(* LS Electric XG5000 project: 210109_AX_FRT_FLR *)
(* PLC NewPLC *)
(* module base 0 slot 0: FEnet:XGL-EFMT(B) (Fast Ethernet 통신 모듈, 전기 Master) *)
(* module base 0 slot 1: FEnet:XGL-EFMT(B) (Fast Ethernet 통신 모듈, 전기 Master) *)
(* module base 0 slot 2: FEnet:XGL-EFMT(B) (Fast Ethernet 통신 모듈, 전기 Master) *)
(* module base 0 slot 3: FEnet:XGL-EFMT(B) (Fast Ethernet 통신 모듈, 전기 Master) *)
(* module base 0 slot 4: FEnet:XGL-EFMT(B) (Fast Ethernet 통신 모듈, 전기 Master) *)
(* module base 0 slot 5: FEnet:XGL-EFMT(B) (Fast Ethernet 통신 모듈, 전기 Master) *)
(* module base 0 slot 6: FEnet:XGL-EFMT(B) (Fast Ethernet 통신 모듈, 전기 Master) *)
(* module base 0 slot 7: FEnet:XGL-EFMT(B) (Fast Ethernet 통신 모듈, 전기 Master) *)
(* module base 0 slot 0: 입력 모듈:XBE-DC16A/B (DC24V 입력, 16점 / DC12/24V 입력, 16점) *)
(* module base 0 slot 1: 입력 모듈:XBE-DC16A/B (DC24V 입력, 16점 / DC12/24V 입력, 16점) *)
(* module base 0 slot 2: 입력 모듈:XBE-DC16A/B (DC24V 입력, 16점 / DC12/24V 입력, 16점) *)
(* module base 0 slot 3: 입력 모듈:XBE-DC16A/B (DC24V 입력, 16점 / DC12/24V 입력, 16점) *)
(* module base 0 slot 4: 출력 모듈:XBE-TN/TP16A (트랜지스터 출력, 16점 (싱크출력/소스출력)) *)
(* module base 0 slot 5: 출력 모듈:XBE-TN/TP16A (트랜지스터 출력, 16점 (싱크출력/소스출력)) *)
(* module base 0 slot 6: 출력 모듈:XBE-TN/TP16A (트랜지스터 출력, 16점 (싱크출력/소스출력)) *)
(* module base 0 slot 7: 출력 모듈:XBE-TN/TP16A (트랜지스터 출력, 16점 (싱크출력/소스출력)) *)
(* module base 0 slot 0: 입력 모듈:XBE-DC16A/B (DC24V 입력, 16점 / DC12/24V 입력, 16점) *)
(* module base 0 slot 1: 입력 모듈:XBE-DC16A/B (DC24V 입력, 16점 / DC12/24V 입력, 16점) *)
(* module base 0 slot 2: 입력 모듈:XBE-DC16A/B (DC24V 입력, 16점 / DC12/24V 입력, 16점) *)
(* module base 0 slot 3: 출력 모듈:XBE-TN/TP16A (트랜지스터 출력, 16점 (싱크출력/소스출력)) *)
(* module base 0 slot 4: 출력 모듈:XBE-TN/TP16A (트랜지스터 출력, 16점 (싱크출력/소스출력)) *)
(* module base 0 slot 0: 입력 모듈:XBE-DC16A/B (DC24V 입력, 16점 / DC12/24V 입력, 16점) *)
(* module base 0 slot 1: 입력 모듈:XBE-DC16A/B (DC24V 입력, 16점 / DC12/24V 입력, 16점) *)
(* module base 0 slot 2: 입력 모듈:XBE-DC16A/B (DC24V 입력, 16점 / DC12/24V 입력, 16점) *)
(* module base 0 slot 3: 출력 모듈:XBE-TN/TP16A (트랜지스터 출력, 16점 (싱크출력/소스출력)) *)
(* module base 0 slot 4: 출력 모듈:XBE-TN/TP16A (트랜지스터 출력, 16점 (싱크출력/소스출력)) *)
(* module base 0 slot 0: 입력 모듈:XBE-DC16A/B (DC24V 입력, 16점 / DC12/24V 입력, 16점) *)
(* module base 0 slot 1: 입력 모듈:XBE-DC16A/B (DC24V 입력, 16점 / DC12/24V 입력, 16점) *)
(* module base 0 slot 2: 입력 모듈:XBE-DC16A/B (DC24V 입력, 16점 / DC12/24V 입력, 16점) *)
(* module base 0 slot 3: 출력 모듈:XBE-TN/TP16A (트랜지스터 출력, 16점 (싱크출력/소스출력)) *)
(* module base 0 slot 4: 출력 모듈:XBE-TN/TP16A (트랜지스터 출력, 16점 (싱크출력/소스출력)) *)
(* module base 0 slot 0: 입력 모듈:XBE-DC16A/B (DC24V 입력, 16점 / DC12/24V 입력, 16점) *)
(* module base 0 slot 1: 출력 모듈:XBE-TN/TP16A (트랜지스터 출력, 16점 (싱크출력/소스출력)) *)
(* module base 0 slot 2: 입력 모듈:XBE-DC16A/B (DC24V 입력, 16점 / DC12/24V 입력, 16점) *)
(* module base 0 slot 3: 출력 모듈:XBE-TN/TP16A (트랜지스터 출력, 16점 (싱크출력/소스출력)) *)
(* module base 0 slot 0: 입력 모듈:XBE-DC16A/B (DC24V 입력, 16점 / DC12/24V 입력, 16점) *)
(* module base 0 slot 1: 입력 모듈:XBE-DC16A/B (DC24V 입력, 16점 / DC12/24V 입력, 16점) *)
(* module base 0 slot 2: 출력 모듈:XBE-TN/TP16A (트랜지스터 출력, 16점 (싱크출력/소스출력)) *)
(* module base 0 slot 3: 입력 모듈:XBE-DC16A/B (DC24V 입력, 16점 / DC12/24V 입력, 16점) *)
(* module base 0 slot 4: 출력 모듈:XBE-TN/TP16A (트랜지스터 출력, 16점 (싱크출력/소스출력)) *)
(* module base 0 slot 0: 입력 모듈:XBE-DC16A/B (DC24V 입력, 16점 / DC12/24V 입력, 16점) *)
(* module base 0 slot 1: 입력 모듈:XBE-DC16A/B (DC24V 입력, 16점 / DC12/24V 입력, 16점) *)
(* module base 0 slot 2: 출력 모듈:XBE-TN/TP16A (트랜지스터 출력, 16점 (싱크출력/소스출력)) *)
(* module base 0 slot 3: 입력 모듈:XBE-DC16A/B (DC24V 입력, 16점 / DC12/24V 입력, 16점) *)
(* module base 0 slot 4: 출력 모듈:XBE-TN/TP16A (트랜지스터 출력, 16점 (싱크출력/소스출력)) *)
(* module base 0 slot 0: 입력 모듈:XBE-DC16A/B (DC24V 입력, 16점 / DC12/24V 입력, 16점) *)
(* module base 0 slot 1: 입력 모듈:XBE-DC16A/B (DC24V 입력, 16점 / DC12/24V 입력, 16점) *)
(* module base 0 slot 2: 입력 모듈:XBE-DC16A/B (DC24V 입력, 16점 / DC12/24V 입력, 16점) *)
(* module base 0 slot 3: 출력 모듈:XBE-TN/TP16A (트랜지스터 출력, 16점 (싱크출력/소스출력)) *)
(* module base 0 slot 4: 출력 모듈:XBE-TN/TP16A (트랜지스터 출력, 16점 (싱크출력/소스출력)) *)
(* module base 0 slot 5: 입력 모듈:XBE-DC16A/B (DC24V 입력, 16점 / DC12/24V 입력, 16점) *)
(* module base 0 slot 6: 출력 모듈:XBE-TN/TP16A (트랜지스터 출력, 16점 (싱크출력/소스출력)) *)
VAR_GLOBAL
    APRON_LH_RACK1_I_막장감지 AT %MW87211.2 : BOOL;
    APRON_LH_RACK1_I_종발이감지1 AT %MW87211.0 : BOOL;
    APRON_LH_RACK1_I_종발이감지2 AT %MW87211.1 : BOOL;
    APRON_LH_RACK2_I_막장감지 AT %MW87211.10 : BOOL;
    APRON_LH_RACK2_I_종발이감지1 AT %MW87211.8 : BOOL;
    APRON_LH_RACK2_I_종발이감지2 AT %MW87211.9 : BOOL;
    APRON_RH_RACK1_I_막장감지 AT %MW87210.2 : BOOL;
    APRON_RH_RACK1_I_종발이감지1 AT %MW87210.0 : BOOL;
    APRON_RH_RACK1_I_종발이감지2 AT %MW87210.1 : BOOL;
    APRON_RH_RACK2_I_막장감지 AT %MW87210.10 : BOOL;
    APRON_RH_RACK2_I_종발이감지1 AT %MW87210.8 : BOOL;
    APRON_RH_RACK2_I_종발이감지2 AT %MW87210.9 : BOOL;
    AWAYS_OFF AT %MW3.0 : BOOL;
    AWAYS_ON AT %MW3.1 : BOOL;
    CARTYPE AT %MW10000 : ARRAY[0..999] OF WORD; (* CARTYPE *)
    CLOCK_BIT_0_1Sec AT %MW0.0 : BOOL;
    CLOCK_BIT_0_2Sec AT %MW0.1 : BOOL;
    CLOCK_BIT_0_4Sec AT %MW0.2 : BOOL;
    CLOCK_BIT_0_5Sec AT %MW0.3 : BOOL;
    CLOCK_BIT_0_8Sec AT %MW0.4 : BOOL;
    CLOCK_BIT_1_0Sec AT %MW0.5 : BOOL;
    CLOCK_BIT_1_6Sec AT %MW0.6 : BOOL;
    CLOCK_BIT_2_0Sec AT %MW0.7 : BOOL;
    DASH_RACK1_I_막장감지 AT %MW87300.2 : BOOL;
    DASH_RACK1_I_종발이감지1 AT %MW87300.0 : BOOL;
    DASH_RACK1_I_종발이감지2 AT %MW87300.1 : BOOL;
    DASH_RACK2_I_막장감지 AT %MW87300.10 : BOOL;
    DASH_RACK2_I_종발이감지1 AT %MW87300.8 : BOOL;
    DASH_RACK2_I_종발이감지2 AT %MW87300.9 : BOOL;
    DASH_RACK3_I_막장감지 AT %MW87301.2 : BOOL;
    DASH_RACK3_I_종발이감지1 AT %MW87301.0 : BOOL;
    DASH_RACK3_I_종발이감지2 AT %MW87301.1 : BOOL;
    DASH_RACK4_I_막장감지 AT %MW87301.10 : BOOL;
    DASH_RACK4_I_종발이감지1 AT %MW87301.8 : BOOL;
    DASH_RACK4_I_종발이감지2 AT %MW87301.9 : BOOL;
    EGIS_EJS : BOOL;
    F_COMPL_I_CYCLE_정지_OK AT %MW83211.7 : BOOL;
    F_COMPL_I_SAFTY_이상 AT %MW83210.14 : BOOL;
    F_COMPL_I_SP1 AT %MW83210.4 : BOOL;
    F_COMPL_I_SP10 AT %MW83211.8 : BOOL;
    F_COMPL_I_SP11 AT %MW83211.9 : BOOL;
    F_COMPL_I_SP12 AT %MW83211.10 : BOOL;
    F_COMPL_I_SP13 AT %MW83211.11 : BOOL;
    F_COMPL_I_SP14 AT %MW83211.12 : BOOL;
    F_COMPL_I_SP15 AT %MW83211.13 : BOOL;
    F_COMPL_I_SP16 AT %MW83211.14 : BOOL;
    F_COMPL_I_SP2 AT %MW83210.5 : BOOL;
    F_COMPL_I_SP3 AT %MW83210.6 : BOOL;
    F_COMPL_I_SP4 AT %MW83210.7 : BOOL;
    F_COMPL_I_SP7 AT %MW83210.10 : BOOL;
    F_COMPL_I_SP8 AT %MW83210.11 : BOOL;
    F_COMPL_I_SP9 AT %MW83210.12 : BOOL;
    F_COMPL_I_SPARE_진입OK AT %MW83211.2 : BOOL;
    F_COMPL_I_도착완료 AT %MW83211.6 : BOOL;
    F_COMPL_I_불간섭 AT %MW83211.0 : BOOL;
    F_COMPL_I_비상정지 AT %MW83210.15 : BOOL;
    F_COMPL_I_수동모드 AT %MW83210.1 : BOOL;
    F_COMPL_I_운전준비 AT %MW83210.0 : BOOL;
    F_COMPL_I_자동_운전중 AT %MW83210.3 : BOOL;
    F_COMPL_I_자동모드 AT %MW83210.2 : BOOL;
    F_COMPL_I_작업완료 AT %MW83211.5 : BOOL;
    F_COMPL_I_진입OK AT %MW83211.1 : BOOL;
    F_COMPL_I_차종수신완료 AT %MW83211.4 : BOOL;
    F_COMPL_I_차종요구 AT %MW83211.3 : BOOL;
    F_COMPL_I_총괄_이상 AT %MW83210.13 : BOOL;
    F_COMPL_I_통신_CHK AT %MW83211.15 : BOOL;
    F_COMPL_I_파트_NONE AT %MW83210.9 : BOOL;
    F_COMPL_I_파트_ON AT %MW83210.8 : BOOL;
    F_COMPL_O_1차종_2차종_3차종 AT %MW93221 : WORD;
    F_COMPL_O_4차종 AT %MW93222 : WORD;
    F_COMPL_O_5차종_6차종_7차종 AT %MW93223 : WORD;
    F_COMPL_O_8차종_9차종 AT %MW93224 : WORD;
    F_COMPL_O_CYCLE_정지_OK AT %MW93211.7 : BOOL;
    F_COMPL_O_SAFTY_이상 AT %MW93210.14 : BOOL;
    F_COMPL_O_SEQ_1 AT %MW93220 : WORD;
    F_COMPL_O_SP1 AT %MW93210.4 : BOOL;
    F_COMPL_O_SP10 AT %MW93211.8 : BOOL;
    F_COMPL_O_SP11 AT %MW93211.9 : BOOL;
    F_COMPL_O_SP12 AT %MW93211.10 : BOOL;
    F_COMPL_O_SP13 AT %MW93211.11 : BOOL;
    F_COMPL_O_SP14 AT %MW93211.12 : BOOL;
    F_COMPL_O_SP15 AT %MW93211.13 : BOOL;
    F_COMPL_O_SP16 AT %MW93211.14 : BOOL;
    F_COMPL_O_SP2 AT %MW93210.5 : BOOL;
    F_COMPL_O_SP3 AT %MW93210.6 : BOOL;
    F_COMPL_O_SP4 AT %MW93210.7 : BOOL;
    F_COMPL_O_SP5 AT %MW93210.8 : BOOL;
    F_COMPL_O_SP6 AT %MW93210.9 : BOOL;
    F_COMPL_O_SP7 AT %MW93210.10 : BOOL;
    F_COMPL_O_SP8 AT %MW93210.11 : BOOL;
    F_COMPL_O_SP9 AT %MW93210.12 : BOOL;
    F_COMPL_O_SPARE_진입OK AT %MW93211.2 : BOOL;
    F_COMPL_O_VIN_NO11 AT %MW93229 : WORD;
    F_COMPL_O_VIN_NO12 AT %MW93230 : WORD;
    F_COMPL_O_VIN_NO13 AT %MW93231 : WORD;
    F_COMPL_O_VIN_NO14 AT %MW93232 : WORD;
    F_COMPL_O_VIN_NO15 AT %MW93233 : WORD;
    F_COMPL_O_도착완료 AT %MW93211.6 : BOOL;
    F_COMPL_O_불간섭 AT %MW93211.0 : BOOL;
    F_COMPL_O_비상정지 AT %MW93210.15 : BOOL;
    F_COMPL_O_수동모드 AT %MW93210.1 : BOOL;
    F_COMPL_O_옵션차종1 AT %MW93225 : WORD;
    F_COMPL_O_옵션차종2 AT %MW93226 : WORD;
    F_COMPL_O_옵션차종3 AT %MW93227 : WORD;
    F_COMPL_O_운영정보 AT %MW93228 : WORD;
    F_COMPL_O_운전준비 AT %MW93210.0 : BOOL;
    F_COMPL_O_자동_운전중 AT %MW93210.3 : BOOL;
    F_COMPL_O_자동모드 AT %MW93210.2 : BOOL;
    F_COMPL_O_작업완료 AT %MW93211.5 : BOOL;
    F_COMPL_O_진입OK AT %MW93211.1 : BOOL;
    F_COMPL_O_차종수신완료 AT %MW93211.4 : BOOL;
    F_COMPL_O_차종요구 AT %MW93211.3 : BOOL;
    F_COMPL_O_총괄_이상 AT %MW93210.13 : BOOL;
    F_COMPL_O_통신_CHK AT %MW93211.15 : BOOL;
    GATE10_M_CP_TRIP AT %MW409.15 : BOOL;
    GATE10_M_GATE_OPEN AT %MW409.13 : BOOL;
    GATE10_M_RESTART AT %MW409.1 : BOOL;
    GATE10_M_도어_잠김 AT %MW409.3 : BOOL;
    GATE10_M_비상정지 AT %MW409.7 : BOOL;
    GATE10_M_이상_리셋 AT %MW409.0 : BOOL;
    GATE10_M_정상 AT %MW409.4 : BOOL;
    GATE10_M_정지_CALL AT %MW409.2 : BOOL;
    GATE10_M_통신_이상 AT %MW409.14 : BOOL;
    GATE11_M_CP_TRIP AT %MW410.15 : BOOL;
    GATE11_M_GATE_OPEN AT %MW410.13 : BOOL;
    GATE11_M_RESTART AT %MW410.1 : BOOL;
    GATE11_M_도어_잠김 AT %MW410.3 : BOOL;
    GATE11_M_비상정지 AT %MW410.7 : BOOL;
    GATE11_M_이상_리셋 AT %MW410.0 : BOOL;
    GATE11_M_정상 AT %MW410.4 : BOOL;
    GATE11_M_정지_CALL AT %MW410.2 : BOOL;
    GATE11_M_통신_이상 AT %MW410.14 : BOOL;
    GATE12_M_CP_TRIP AT %MW411.15 : BOOL;
    GATE12_M_GATE_OPEN AT %MW411.13 : BOOL;
    GATE12_M_RESTART AT %MW411.1 : BOOL;
    GATE12_M_도어_잠김 AT %MW411.3 : BOOL;
    GATE12_M_비상정지 AT %MW411.7 : BOOL;
    GATE12_M_이상_리셋 AT %MW411.0 : BOOL;
    GATE12_M_정상 AT %MW411.4 : BOOL;
    GATE12_M_정지_CALL AT %MW411.2 : BOOL;
    GATE12_M_통신_이상 AT %MW411.14 : BOOL;
    GATE_10_M_GATE_OPEN_보조 AT %MW409.12 : BOOL;
    GATE_11_M_GATE_OPEN_보조 AT %MW410.12 : BOOL;
    GATE_12_M_GATE_OPEN_보조 AT %MW411.12 : BOOL;
    GB10_7_10_PLC_BOX_CP_TRIP AT %MW87100.15 : BOOL; (* 입력 접점 15 *)
    GB10_EPB_비상정지1 AT %MW87102.0 : BOOL; (* 입력 접점 00 *)
    GB10_EPB_비상정지2 AT %MW87102.1 : BOOL; (* 입력 접점 01 *)
    GB10_GATE_LOCK_SW_열림1 AT %MW87102.8 : BOOL; (* 입력 접점 08 *)
    GB10_GATE_LOCK_SW_열림2 AT %MW87102.9 : BOOL; (* 입력 접점 09 *)
    GB10_PBL_CYCLE_정지 AT %MW87100.1 : BOOL; (* 입력 접점 01 *)
    GB10_PBL_CYCLE_정지_LP AT %MW97101.1 : BOOL; (* 출력 접점 01 *)
    GB10_PBL_자동_운전 AT %MW87100.0 : BOOL; (* 입력 접점 00 *)
    GB10_PBL_자동_운전_LP AT %MW97101.0 : BOOL; (* 출력 접점 00 *)
    GB10_PB_이상_리셋 AT %MW87100.2 : BOOL; (* 입력 접점 02 *)
    GB10_SAFETY_DOOR_UNLOOK1 AT %MW97103.0 : BOOL; (* 출력 접점 00 *)
    GB10_SAFETY_DOOR_UNLOOK2 AT %MW97103.1 : BOOL; (* 출력 접점 01 *)
    GB10_TL_GREEN_LAMP AT %MW97101.9 : BOOL; (* 출력 접점 09 *)
    GB10_TL_RED_LAMP AT %MW97101.8 : BOOL; (* 출력 접점 08 *)
    HMI_M_SEL_MOD_S101 AT %MW6.1 : BOOL;
    HMI_M_SEL_MOD_S102 AT %MW6.2 : BOOL;
    HMI_M_SEL_MOD_S103 AT %MW6.3 : BOOL;
    HMI_M_SEL_MOD_STN AT %MW6.0 : BOOL;
    HMI_M_매칭_R102_1_S101 AT %MW70.1 : BOOL;
    HMI_M_매칭_S101_R102_1 AT %MW70.0 : BOOL;
    HMI_M_매칭선택 AT %MW70 : WORD;
    HMI_M_매칭차종_DATA_OK AT %MW9.9 : BOOL;
    HMI_M_매칭차종_복사_ON AT %MW9.6 : BOOL;
    HMI_M_매칭차종_복사_SET AT %MW9.8 : BOOL;
    HMI_M_매칭차종_복사_가능 AT %MW9.7 : BOOL;
    HMI_M_선택_MOD_CARR AT %MW12 : WORD;
    HMI_M_선택_MOD_PROF AT %MW13 : WORD;
    HMI_M_차종매칭 AT %MW50 : ARRAY[0..19] OF WORD;
    HMI_M_차종매칭_SEQ AT %MW50 : WORD;
    HMI_M_차종매칭_VIN_NO_1_2 AT %MW61 : WORD;
    HMI_M_차종매칭_VIN_NO_3_4 AT %MW62 : WORD;
    HMI_M_차종매칭_VIN_NO_5_6 AT %MW63 : WORD;
    HMI_M_차종매칭_VIN_NO_7_8 AT %MW64 : WORD;
    HMI_M_차종매칭_VIN_NO_9_10 AT %MW65 : WORD;
    HMI_M_차종매칭_차종1_AX AT %MW51.0 : BOOL;
    HMI_M_차종매칭_차종1_B AT %MW51.1 : BOOL;
    HMI_M_차종매칭_차종1_C AT %MW51.2 : BOOL;
    HMI_M_차종매칭_차종1_D AT %MW51.3 : BOOL;
    HMI_M_차종매칭_차종1_E AT %MW51.4 : BOOL;
    HMI_M_차종매칭_차종1_F AT %MW51.5 : BOOL;
    HMI_M_차종매칭_차종1_G AT %MW51.6 : BOOL;
    HMI_M_차종매칭_차종1_H AT %MW51.7 : BOOL;
    HMI_M_차종매칭_차종2_3DR AT %MW51.8 : BOOL;
    HMI_M_차종매칭_차종2_4DR AT %MW51.9 : BOOL;
    HMI_M_차종매칭_차종2_5DR AT %MW51.10 : BOOL;
    HMI_M_차종매칭_차종2_SP1 AT %MW51.12 : BOOL;
    HMI_M_차종매칭_차종2_SP2 AT %MW51.13 : BOOL;
    HMI_M_차종매칭_차종2_WGN AT %MW51.11 : BOOL;
    HMI_M_차종매칭_차종3_LHD AT %MW51.14 : BOOL;
    HMI_M_차종매칭_차종3_RHD AT %MW51.15 : BOOL;
    HMI_M_차종매칭_차종4_EEC AT %MW52.3 : BOOL;
    HMI_M_차종매칭_차종4_SP1 AT %MW52.8 : BOOL;
    HMI_M_차종매칭_차종4_SP2 AT %MW52.9 : BOOL;
    HMI_M_차종매칭_차종4_SP3 AT %MW52.11 : BOOL;
    HMI_M_차종매칭_차종4_SP4 AT %MW52.12 : BOOL;
    HMI_M_차종매칭_차종4_SP5 AT %MW52.13 : BOOL;
    HMI_M_차종매칭_차종4_SP6 AT %MW52.14 : BOOL;
    HMI_M_차종매칭_차종4_SP7 AT %MW52.15 : BOOL;
    HMI_M_차종매칭_차종4_내수 AT %MW52.0 : BOOL;
    HMI_M_차종매칭_차종4_러시아 AT %MW52.10 : BOOL;
    HMI_M_차종매칭_차종4_북미 AT %MW52.2 : BOOL;
    HMI_M_차종매칭_차종4_브라질 AT %MW52.7 : BOOL;
    HMI_M_차종매칭_차종4_수출 AT %MW52.1 : BOOL;
    HMI_M_차종매칭_차종4_중국 AT %MW52.6 : BOOL;
    HMI_M_차종매칭_차종4_중동 AT %MW52.5 : BOOL;
    HMI_M_차종매칭_차종4_호주 AT %MW52.4 : BOOL;
    HMI_M_차종매칭_차종5_AT AT %MW53.1 : BOOL;
    HMI_M_차종매칭_차종5_MT AT %MW53.0 : BOOL;
    HMI_M_차종매칭_차종5_SP1 AT %MW53.2 : BOOL;
    HMI_M_차종매칭_차종6_DSROOF AT %MW53.6 : BOOL;
    HMI_M_차종매칭_차종6_SP1 AT %MW53.7 : BOOL;
    HMI_M_차종매칭_차종6_썬루프 AT %MW53.4 : BOOL;
    HMI_M_차종매칭_차종6_일반루프 AT %MW53.3 : BOOL;
    HMI_M_차종매칭_차종6_파노라마루프 AT %MW53.5 : BOOL;
    HMI_M_차종매칭_차종7_DSL AT %MW53.9 : BOOL;
    HMI_M_차종매칭_차종7_GSL AT %MW53.8 : BOOL;
    HMI_M_차종매칭_차종7_SP1 AT %MW53.10 : BOOL;
    HMI_M_차종매칭_차종7_SP2 AT %MW53.11 : BOOL;
    HMI_M_차종매칭_차종7_SP3 AT %MW53.12 : BOOL;
    HMI_M_차종매칭_차종7_SP4 AT %MW53.13 : BOOL;
    HMI_M_차종매칭_차종7_SP5 AT %MW53.14 : BOOL;
    HMI_M_차종매칭_차종7_SP6 AT %MW53.15 : BOOL;
    HMI_M_차종매칭_차종8_2WD AT %MW54.0 : BOOL;
    HMI_M_차종매칭_차종8_4WD AT %MW54.1 : BOOL;
    HMI_M_차종매칭_차종8_SP1 AT %MW54.2 : BOOL;
    HMI_M_차종매칭_차종9_MPI AT %MW54.3 : BOOL;
    HMI_M_차종매칭_차종9_SP1 AT %MW54.5 : BOOL;
    HMI_M_차종매칭_차종9_SP10 AT %MW54.14 : BOOL;
    HMI_M_차종매칭_차종9_SP11 AT %MW54.15 : BOOL;
    HMI_M_차종매칭_차종9_SP2 AT %MW54.6 : BOOL;
    HMI_M_차종매칭_차종9_SP3 AT %MW54.7 : BOOL;
    HMI_M_차종매칭_차종9_SP4 AT %MW54.8 : BOOL;
    HMI_M_차종매칭_차종9_SP5 AT %MW54.9 : BOOL;
    HMI_M_차종매칭_차종9_SP6 AT %MW54.10 : BOOL;
    HMI_M_차종매칭_차종9_SP7 AT %MW54.11 : BOOL;
    HMI_M_차종매칭_차종9_SP8 AT %MW54.12 : BOOL;
    HMI_M_차종매칭_차종9_SP9 AT %MW54.13 : BOOL;
    HMI_M_차종매칭_차종9_T_GDI AT %MW54.4 : BOOL;
    HMI_M_차종매칭_차종_AS AT %MW60.9 : BOOL;
    HMI_M_차종매칭_차종_OPT1_R_RACK_무 AT %MW55.3 : BOOL;
    HMI_M_차종매칭_차종_OPT1_R_RACK_유 AT %MW55.2 : BOOL;
    HMI_M_차종매칭_차종_OPT1_SP1 AT %MW55.10 : BOOL;
    HMI_M_차종매칭_차종_OPT1_SP2 AT %MW55.11 : BOOL;
    HMI_M_차종매칭_차종_OPT1_SP3 AT %MW55.12 : BOOL;
    HMI_M_차종매칭_차종_OPT1_SP4 AT %MW55.13 : BOOL;
    HMI_M_차종매칭_차종_OPT1_SP5 AT %MW55.14 : BOOL;
    HMI_M_차종매칭_차종_OPT1_SP6 AT %MW55.15 : BOOL;
    HMI_M_차종매칭_차종_OPT1_S_REP_EATER_무 AT %MW55.7 : BOOL;
    HMI_M_차종매칭_차종_OPT1_S_REP_EATER_유 AT %MW55.6 : BOOL;
    HMI_M_차종매칭_차종_OPT1_VAN_무 AT %MW55.9 : BOOL;
    HMI_M_차종매칭_차종_OPT1_VAN_유 AT %MW55.8 : BOOL;
    HMI_M_차종매칭_차종_OPT1_슬라이딩_무 AT %MW55.1 : BOOL;
    HMI_M_차종매칭_차종_OPT1_슬라이딩_유 AT %MW55.0 : BOOL;
    HMI_M_차종매칭_차종_OPT1_폴딩_무 AT %MW55.5 : BOOL;
    HMI_M_차종매칭_차종_OPT1_폴딩_유 AT %MW55.4 : BOOL;
    HMI_M_차종매칭_차종_OPT2_SP_WORD1 AT %MW56 : WORD;
    HMI_M_차종매칭_차종_OPT3_SP_WORD2 AT %MW57 : WORD;
    HMI_M_차종매칭_차종_OPT4_SP_WORD3 AT %MW58 : WORD;
    HMI_M_차종매칭_차종_OPT5_SP_WORD4 AT %MW59 : WORD;
    HMI_M_차종매칭_차종_SP1 AT %MW60.0 : BOOL;
    HMI_M_차종매칭_차종_SP2 AT %MW60.1 : BOOL;
    HMI_M_차종매칭_차종_SP3 AT %MW60.2 : BOOL;
    HMI_M_차종매칭_차종_SP4 AT %MW60.3 : BOOL;
    HMI_M_차종매칭_차종_SP5 AT %MW60.4 : BOOL;
    HMI_M_차종매칭_차종_SP6 AT %MW60.5 : BOOL;
    HMI_M_차종매칭_차종_SP7 AT %MW60.6 : BOOL;
    HMI_M_차종매칭_차종_SP8 AT %MW60.7 : BOOL;
    HMI_M_차종매칭_차종_SP9 AT %MW60.15 : BOOL;
    HMI_M_차종매칭_차종_공대차 AT %MW60.12 : BOOL;
    HMI_M_차종매칭_차종_공차 AT %MW60.10 : BOOL;
    HMI_M_차종매칭_차종_불량대차 AT %MW60.13 : BOOL;
    HMI_M_차종매칭_차종_불량차 AT %MW60.11 : BOOL;
    HMI_M_차종매칭_차종_비축 AT %MW60.8 : BOOL;
    HMI_M_차종매칭_차종_취출대차 AT %MW60.14 : BOOL;
    HMI_M_차종수정 AT %MW10 : ARRAY[0..19] OF WORD;
    HMI_M_차종수정_DATA_OK AT %MW9.0 : BOOL;
    HMI_M_차종수정_RESET AT %MW9.2 : BOOL;
    HMI_M_차종수정_SEQ AT %MW10 : WORD;
    HMI_M_차종수정_SET AT %MW9.1 : BOOL;
    HMI_M_차종수정_VIN_NO_1_2 AT %MW21 : WORD;
    HMI_M_차종수정_VIN_NO_3_4 AT %MW22 : WORD;
    HMI_M_차종수정_VIN_NO_5_6 AT %MW23 : WORD;
    HMI_M_차종수정_VIN_NO_7_8 AT %MW24 : WORD;
    HMI_M_차종수정_VIN_NO_9_10 AT %MW25 : WORD;
    HMI_M_차종수정_차종1_AX AT %MW11.0 : BOOL;
    HMI_M_차종수정_차종1_B AT %MW11.1 : BOOL;
    HMI_M_차종수정_차종1_C AT %MW11.2 : BOOL;
    HMI_M_차종수정_차종1_D AT %MW11.3 : BOOL;
    HMI_M_차종수정_차종1_E AT %MW11.4 : BOOL;
    HMI_M_차종수정_차종1_F AT %MW11.5 : BOOL;
    HMI_M_차종수정_차종1_G AT %MW11.6 : BOOL;
    HMI_M_차종수정_차종1_H AT %MW11.7 : BOOL;
    HMI_M_차종수정_차종2_3DR AT %MW11.8 : BOOL;
    HMI_M_차종수정_차종2_4DR AT %MW11.9 : BOOL;
    HMI_M_차종수정_차종2_5DR AT %MW11.10 : BOOL;
    HMI_M_차종수정_차종2_SP1 AT %MW11.12 : BOOL;
    HMI_M_차종수정_차종2_SP2 AT %MW11.13 : BOOL;
    HMI_M_차종수정_차종2_WGN AT %MW11.11 : BOOL;
    HMI_M_차종수정_차종3_LHD AT %MW11.14 : BOOL;
    HMI_M_차종수정_차종3_RHD AT %MW11.15 : BOOL;
    HMI_M_차종수정_차종4_EEC AT %MW12.3 : BOOL;
    HMI_M_차종수정_차종4_SP1 AT %MW12.8 : BOOL;
    HMI_M_차종수정_차종4_SP2 AT %MW12.9 : BOOL;
    HMI_M_차종수정_차종4_SP3 AT %MW12.11 : BOOL;
    HMI_M_차종수정_차종4_SP4 AT %MW12.12 : BOOL;
    HMI_M_차종수정_차종4_SP5 AT %MW12.13 : BOOL;
    HMI_M_차종수정_차종4_SP6 AT %MW12.14 : BOOL;
    HMI_M_차종수정_차종4_SP7 AT %MW12.15 : BOOL;
    HMI_M_차종수정_차종4_내수 AT %MW12.0 : BOOL;
    HMI_M_차종수정_차종4_러시아 AT %MW12.10 : BOOL;
    HMI_M_차종수정_차종4_북미 AT %MW12.2 : BOOL;
    HMI_M_차종수정_차종4_브라질 AT %MW12.7 : BOOL;
    HMI_M_차종수정_차종4_수출 AT %MW12.1 : BOOL;
    HMI_M_차종수정_차종4_중국 AT %MW12.6 : BOOL;
    HMI_M_차종수정_차종4_중동 AT %MW12.5 : BOOL;
    HMI_M_차종수정_차종4_호주 AT %MW12.4 : BOOL;
    HMI_M_차종수정_차종5_AT AT %MW13.1 : BOOL;
    HMI_M_차종수정_차종5_MT AT %MW13.0 : BOOL;
    HMI_M_차종수정_차종5_SP1 AT %MW13.2 : BOOL;
    HMI_M_차종수정_차종6_DSROOF AT %MW13.6 : BOOL;
    HMI_M_차종수정_차종6_SP1 AT %MW13.7 : BOOL;
    HMI_M_차종수정_차종6_썬루프 AT %MW13.4 : BOOL;
    HMI_M_차종수정_차종6_일반루프 AT %MW13.3 : BOOL;
    HMI_M_차종수정_차종6_파노라마루프 AT %MW13.5 : BOOL;
    HMI_M_차종수정_차종7_DSL AT %MW13.9 : BOOL;
    HMI_M_차종수정_차종7_GSL AT %MW13.8 : BOOL;
    HMI_M_차종수정_차종7_SP1 AT %MW13.10 : BOOL;
    HMI_M_차종수정_차종7_SP2 AT %MW13.11 : BOOL;
    HMI_M_차종수정_차종7_SP3 AT %MW13.12 : BOOL;
    HMI_M_차종수정_차종7_SP4 AT %MW13.13 : BOOL;
    HMI_M_차종수정_차종7_SP5 AT %MW13.14 : BOOL;
    HMI_M_차종수정_차종7_SP6 AT %MW13.15 : BOOL;
    HMI_M_차종수정_차종8_2WD AT %MW14.0 : BOOL;
    HMI_M_차종수정_차종8_4WD AT %MW14.1 : BOOL;
    HMI_M_차종수정_차종8_SP1 AT %MW14.2 : BOOL;
    HMI_M_차종수정_차종9_MPI AT %MW14.3 : BOOL;
    HMI_M_차종수정_차종9_SP1 AT %MW14.5 : BOOL;
    HMI_M_차종수정_차종9_SP10 AT %MW14.14 : BOOL;
    HMI_M_차종수정_차종9_SP11 AT %MW14.15 : BOOL;
    HMI_M_차종수정_차종9_SP2 AT %MW14.6 : BOOL;
    HMI_M_차종수정_차종9_SP3 AT %MW14.7 : BOOL;
    HMI_M_차종수정_차종9_SP4 AT %MW14.8 : BOOL;
    HMI_M_차종수정_차종9_SP5 AT %MW14.9 : BOOL;
    HMI_M_차종수정_차종9_SP6 AT %MW14.10 : BOOL;
    HMI_M_차종수정_차종9_SP7 AT %MW14.11 : BOOL;
    HMI_M_차종수정_차종9_SP8 AT %MW14.12 : BOOL;
    HMI_M_차종수정_차종9_SP9 AT %MW14.13 : BOOL;
    HMI_M_차종수정_차종9_T_GDI AT %MW14.4 : BOOL;
    HMI_M_차종수정_차종_AS AT %MW20.9 : BOOL;
    HMI_M_차종수정_차종_OPT1_R_RACK_무 AT %MW15.3 : BOOL;
    HMI_M_차종수정_차종_OPT1_R_RACK_유 AT %MW15.2 : BOOL;
    HMI_M_차종수정_차종_OPT1_SP1 AT %MW15.10 : BOOL;
    HMI_M_차종수정_차종_OPT1_SP2 AT %MW15.11 : BOOL;
    HMI_M_차종수정_차종_OPT1_SP3 AT %MW15.12 : BOOL;
    HMI_M_차종수정_차종_OPT1_SP4 AT %MW15.13 : BOOL;
    HMI_M_차종수정_차종_OPT1_SP5 AT %MW15.14 : BOOL;
    HMI_M_차종수정_차종_OPT1_SP6 AT %MW15.15 : BOOL;
    HMI_M_차종수정_차종_OPT1_S_REP_EATER_무 AT %MW15.7 : BOOL;
    HMI_M_차종수정_차종_OPT1_S_REP_EATER_유 AT %MW15.6 : BOOL;
    HMI_M_차종수정_차종_OPT1_VAN_무 AT %MW15.9 : BOOL;
    HMI_M_차종수정_차종_OPT1_VAN_유 AT %MW15.8 : BOOL;
    HMI_M_차종수정_차종_OPT1_슬라이딩_무 AT %MW15.1 : BOOL;
    HMI_M_차종수정_차종_OPT1_슬라이딩_유 AT %MW15.0 : BOOL;
    HMI_M_차종수정_차종_OPT1_폴딩_무 AT %MW15.5 : BOOL;
    HMI_M_차종수정_차종_OPT1_폴딩_유 AT %MW15.4 : BOOL;
    HMI_M_차종수정_차종_OPT2_SP_WORD1 AT %MW16 : WORD;
    HMI_M_차종수정_차종_OPT3_SP_WORD2 AT %MW17 : WORD;
    HMI_M_차종수정_차종_OPT4_SP_WORD3 AT %MW18 : WORD;
    HMI_M_차종수정_차종_OPT5_SP_WORD4 AT %MW19 : WORD;
    HMI_M_차종수정_차종_SP1 AT %MW20.0 : BOOL;
    HMI_M_차종수정_차종_SP2 AT %MW20.1 : BOOL;
    HMI_M_차종수정_차종_SP3 AT %MW20.2 : BOOL;
    HMI_M_차종수정_차종_SP4 AT %MW20.3 : BOOL;
    HMI_M_차종수정_차종_SP5 AT %MW20.4 : BOOL;
    HMI_M_차종수정_차종_SP6 AT %MW20.5 : BOOL;
    HMI_M_차종수정_차종_SP7 AT %MW20.6 : BOOL;
    HMI_M_차종수정_차종_SP8 AT %MW20.7 : BOOL;
    HMI_M_차종수정_차종_SP9 AT %MW20.15 : BOOL;
    HMI_M_차종수정_차종_공대차 AT %MW20.12 : BOOL;
    HMI_M_차종수정_차종_공차 AT %MW20.10 : BOOL;
    HMI_M_차종수정_차종_불량대차 AT %MW20.13 : BOOL;
    HMI_M_차종수정_차종_불량차 AT %MW20.11 : BOOL;
    HMI_M_차종수정_차종_비축 AT %MW20.8 : BOOL;
    HMI_M_차종수정_차종_취출대차 AT %MW20.14 : BOOL;
    HMI_M_차종수정가능_OK AT %MW9.4 : BOOL;
    HMI_M_차종수정가능_SEL AT %MW9.3 : BOOL;
    HMI_M_현재표출_차종 AT %MW30 : ARRAY[0..19] OF WORD;
    HMI_차종매칭_공정선택 AT %MW8 : WORD;
    HMI_차종수정_공정선택 AT %MW7 : WORD;
    MCP_DISPLAY_CP_TRIP AT %MW87632.5 : BOOL; (* 입력 접점 05 *)
    MCP_EPB_비상정지1 AT %MW87635.0 : BOOL; (* 입력 접점 00 *)
    MCP_EPB_비상정지2 AT %MW87635.1 : BOOL; (* 입력 접점 01 *)
    MCP_HMI_CP_TRIP AT %MW87632.4 : BOOL; (* 입력 접점 04 *)
    MCP_HUB_CP_TRIP AT %MW87632.0 : BOOL; (* 입력 접점 00 *)
    MCP_INPUT_PWR_CP_TRIP AT %MW87632.2 : BOOL; (* 입력 접점 02 *)
    MCP_KSW_MES_OFF AT %MW87631.4 : BOOL; (* 입력 접점 04 *)
    MCP_KSW_MES_ON AT %MW87631.5 : BOOL; (* 입력 접점 05 *)
    MCP_MC1_OUTPUT_PWR_ON AT %MW97636.0 : BOOL; (* 출력 접점 00 *)
    MCP_M_CP_OFF_이상 AT %MW351.0 : BOOL;
    MCP_M_DISPLAY_CP_TRIP AT %MW351.6 : BOOL;
    MCP_M_FAN_이상 AT %MW352.5 : BOOL;
    MCP_M_HMI_CP_TRIP AT %MW351.7 : BOOL;
    MCP_M_HUB_CP_TRIP AT %MW351.1 : BOOL;
    MCP_M_INPUT_CP_TRIP AT %MW351.3 : BOOL;
    MCP_M_OUTPUT_CP_TRIP AT %MW351.4 : BOOL;
    MCP_M_OUTPUT_MC_OFF AT %MW350.11 : BOOL;
    MCP_M_OUTPUT_MC_ON AT %MW350.10 : BOOL;
    MCP_M_OUTPUT_MC_이상 AT %MW354.8 : BOOL;
    MCP_M_PROFI_PWR_CP_TRIP AT %MW351.5 : BOOL;
    MCP_M_PS1_DC_LOW AT %MW353.6 : BOOL;
    MCP_M_PS2_DC_LOW AT %MW353.7 : BOOL;
    MCP_M_PS3_DC_LOW AT %MW353.8 : BOOL;
    MCP_M_PS4_DC_LOW AT %MW353.9 : BOOL;
    MCP_M_PS_DC_LOW AT %MW353.5 : BOOL;
    MCP_M_SAG1_1_이상 AT %MW352.1 : BOOL;
    MCP_M_SAG1_2_이상 AT %MW352.2 : BOOL;
    MCP_M_SAG_이상 AT %MW352.0 : BOOL;
    MCP_M_SPD_이상 AT %MW354.0 : BOOL;
    MCP_M_램프_테스트 AT %MW350.6 : BOOL;
    MCP_M_부저_정지 AT %MW350.5 : BOOL;
    MCP_M_비상정지 AT %MW350.7 : BOOL;
    MCP_M_수동_모드 AT %MW350.1 : BOOL;
    MCP_M_운전준비_ON AT %MW350.0 : BOOL;
    MCP_M_이상_리셋 AT %MW350.4 : BOOL;
    MCP_M_자동_START AT %MW350.3 : BOOL;
    MCP_M_자동_모드 AT %MW350.2 : BOOL;
    MCP_M_통신_CP_TRIP AT %MW351.2 : BOOL;
    MCP_M_통신_이상 AT %MW352.8 : BOOL;
    MCP_OUTPUT_PWR_CP_TRIP AT %MW87632.3 : BOOL; (* 입력 접점 03 *)
    MCP_PBL_101_자동_운전 AT %MW87630.4 : BOOL; (* 입력 접점 04 *)
    MCP_PBL_101_자동_운전_LP AT %MW97633.1 : BOOL; (* 출력 접점 01 *)
    MCP_PBL_102_자동_운전 AT %MW87630.7 : BOOL; (* 입력 접점 07 *)
    MCP_PBL_102_자동_운전_LP AT %MW97633.2 : BOOL; (* 출력 접점 02 *)
    MCP_PBL_103_4_자동_운전 AT %MW87630.10 : BOOL; (* 입력 접점 10 *)
    MCP_PBL_103_4_자동_운전_LP AT %MW97633.3 : BOOL; (* 출력 접점 03 *)
    MCP_PBL_운전준비_ON AT %MW87630.0 : BOOL; (* 입력 접점 00 *)
    MCP_PBL_운전준비_ON_LP AT %MW97633.0 : BOOL; (* 출력 접점 00 *)
    MCP_PB_이상_리셋 AT %MW87630.1 : BOOL; (* 입력 접점 01 *)
    MCP_PS1_DC_OK AT %MW87631.12 : BOOL; (* 입력 접점 12 *)
    MCP_PS2_DC_OK AT %MW87631.13 : BOOL; (* 입력 접점 13 *)
    MCP_PS3_DC_OK AT %MW87631.14 : BOOL; (* 입력 접점 14 *)
    MCP_SAFTY_MC_ON AT %MW87632.9 : BOOL; (* 입력 접점 09 *)
    MCP_SPB_램프_테스트 AT %MW87631.2 : BOOL; (* 입력 접점 02 *)
    MCP_SPB_부저_정지 AT %MW87631.3 : BOOL; (* 입력 접점 03 *)
    MCP_SPK_MEL1 AT %MW97633.8 : BOOL; (* 출력 접점 08 *)
    MCP_SSP_101_수동_선택 AT %MW87630.2 : BOOL; (* 입력 접점 02 *)
    MCP_SSP_101_자동_선택 AT %MW87630.3 : BOOL; (* 입력 접점 03 *)
    MCP_SSP_102_수동_선택 AT %MW87630.5 : BOOL; (* 입력 접점 05 *)
    MCP_SSP_102_자동_선택 AT %MW87630.6 : BOOL; (* 입력 접점 06 *)
    MCP_SSP_103_4_수동_선택 AT %MW87630.8 : BOOL; (* 입력 접점 08 *)
    MCP_SSP_103_4_자동_선택 AT %MW87630.9 : BOOL; (* 입력 접점 09 *)
    MCP_TL_GREEN_LAMP AT %MW97633.6 : BOOL; (* 출력 접점 06 *)
    MCP_TL_RED_LAMP AT %MW97633.4 : BOOL; (* 출력 접점 04 *)
    MCP_TL_YELLOW_LAMP AT %MW97633.5 : BOOL; (* 출력 접점 05 *)
    MCP_타워_부저 AT %MW97633.7 : BOOL; (* 출력 접점 07 *)
    MCP_통신_CP_TRIP AT %MW87632.1 : BOOL; (* 입력 접점 01 *)
    OTR_RACK1_I_막장감지 AT %MW87020.2 : BOOL;
    OTR_RACK1_I_종발이감지1 AT %MW87020.0 : BOOL;
    OTR_RACK1_I_종발이감지2 AT %MW87020.1 : BOOL;
    OTR_RACK2_I_막장감지 AT %MW87020.10 : BOOL;
    OTR_RACK2_I_종발이감지1 AT %MW87020.8 : BOOL;
    OTR_RACK2_I_종발이감지2 AT %MW87020.9 : BOOL;
    PWR_FAN_이상 AT %MW352.6 : BOOL;
    PWR_SAG1_DSUB1_NOMAL1 AT %MW87631.10 : BOOL; (* 입력 접점 10 *)
    PWR_SAG1_DSUB8_NOMAL2 AT %MW87631.11 : BOOL; (* 입력 접점 11 *)
    PWR_SPD1_NOMAL AT %MW87631.8 : BOOL; (* 입력 접점 08 *)
    R101_1_1_I_RB_0_5_COMM_CHK AT %MW84043.14 : BOOL;
    R101_1_1_I_RB_10차_간섭무 AT %MW84041.9 : BOOL;
    R101_1_1_I_RB_11차_간섭무 AT %MW84041.10 : BOOL;
    R101_1_1_I_RB_12차_간섭무 AT %MW84041.11 : BOOL;
    R101_1_1_I_RB_1차_간섭무 AT %MW84041.0 : BOOL;
    R101_1_1_I_RB_1차_작업완료 AT %MW84040.9 : BOOL;
    R101_1_1_I_RB_2차_간섭무 AT %MW84041.1 : BOOL;
    R101_1_1_I_RB_2차_작업완료 AT %MW84040.10 : BOOL;
    R101_1_1_I_RB_3차_간섭무 AT %MW84041.2 : BOOL;
    R101_1_1_I_RB_3차_작업완료 AT %MW84040.11 : BOOL;
    R101_1_1_I_RB_4차_간섭무 AT %MW84041.3 : BOOL;
    R101_1_1_I_RB_4차_작업완료 AT %MW84040.12 : BOOL;
    R101_1_1_I_RB_5차_간섭무 AT %MW84041.4 : BOOL;
    R101_1_1_I_RB_5차_작업완료 AT %MW84040.13 : BOOL;
    R101_1_1_I_RB_6차_간섭무 AT %MW84041.5 : BOOL;
    R101_1_1_I_RB_6차_작업완료 AT %MW84040.14 : BOOL;
    R101_1_1_I_RB_7차_간섭무 AT %MW84041.6 : BOOL;
    R101_1_1_I_RB_7차_작업완료 AT %MW84040.15 : BOOL;
    R101_1_1_I_RB_8차_간섭무 AT %MW84041.7 : BOOL;
    R101_1_1_I_RB_9차_간섭무 AT %MW84041.8 : BOOL;
    R101_1_1_I_RB_AB_NORMAL_선택 AT %MW84040.6 : BOOL;
    R101_1_1_I_RB_GUN1_FIXED_TIP AT %MW84047 : WORD;
    R101_1_1_I_RB_GUN1_MOVING_TIP AT %MW84046 : WORD;
    R101_1_1_I_RB_GUN2_FIXED_TIP AT %MW84049 : WORD;
    R101_1_1_I_RB_GUN2_MOVING_TIP AT %MW84048 : WORD;
    R101_1_1_I_RB_INPUT AT %MW84040 : ARRAY[0..3] OF WORD;
    R101_1_1_I_RB_LS_이상 AT %MW84042.11 : BOOL;
    R101_1_1_I_RB_MOTOR_MC_ON AT %MW84043.15 : BOOL;
    R101_1_1_I_RB_MUTUAL_INT1 AT %MW84043.0 : BOOL;
    R101_1_1_I_RB_MUTUAL_INT2 AT %MW84043.1 : BOOL;
    R101_1_1_I_RB_MUTUAL_INT3 AT %MW84043.2 : BOOL;
    R101_1_1_I_RB_MUTUAL_INT4 AT %MW84043.3 : BOOL;
    R101_1_1_I_RB_MUTUAL_INT5 AT %MW84043.4 : BOOL;
    R101_1_1_I_RB_MUTUAL_INT6 AT %MW84043.5 : BOOL;
    R101_1_1_I_RB_MUTUAL_INT7 AT %MW84043.6 : BOOL;
    R101_1_1_I_RB_MUTUAL_INT8 AT %MW84043.7 : BOOL;
    R101_1_1_I_RB_PLT_UNLOAD_완료 AT %MW84043.11 : BOOL;
    R101_1_1_I_RB_PLT_최종UNLOAD_완료 AT %MW84043.12 : BOOL;
    R101_1_1_I_RB_PROG_ECHO_1 AT %MW84042.0 : BOOL;
    R101_1_1_I_RB_PROG_ECHO_128 AT %MW84042.7 : BOOL;
    R101_1_1_I_RB_PROG_ECHO_16 AT %MW84042.4 : BOOL;
    R101_1_1_I_RB_PROG_ECHO_2 AT %MW84042.1 : BOOL;
    R101_1_1_I_RB_PROG_ECHO_32 AT %MW84042.5 : BOOL;
    R101_1_1_I_RB_PROG_ECHO_4 AT %MW84042.2 : BOOL;
    R101_1_1_I_RB_PROG_ECHO_64 AT %MW84042.6 : BOOL;
    R101_1_1_I_RB_PROG_ECHO_8 AT %MW84042.3 : BOOL;
    R101_1_1_I_RB_SP3_8 AT %MW84043.8 : BOOL;
    R101_1_1_I_RB_SP3_9 AT %MW84043.9 : BOOL;
    R101_1_1_I_RB_SPARE_WORD_4 AT %MW84044 : WORD;
    R101_1_1_I_RB_SP_1_12 AT %MW84041.12 : BOOL;
    R101_1_1_I_RB_SP_1_13 AT %MW84041.13 : BOOL;
    R101_1_1_I_RB_SP_1_14 AT %MW84041.14 : BOOL;
    R101_1_1_I_RB_SP_1_15 AT %MW84041.15 : BOOL;
    R101_1_1_I_RB_TC_이상 AT %MW84042.8 : BOOL;
    R101_1_1_I_RB_TIP_CHANGE AT %MW84043.13 : BOOL;
    R101_1_1_I_RB_TIP_DRESSING AT %MW84040.7 : BOOL;
    R101_1_1_I_RB__PLT_카운터리셋완료 AT %MW84043.10 : BOOL;
    R101_1_1_I_RB_공기압_이상 AT %MW84042.9 : BOOL;
    R101_1_1_I_RB_냉각수_이상 AT %MW84042.10 : BOOL;
    R101_1_1_I_RB_비상정지_NC AT %MW84040.8 : BOOL;
    R101_1_1_I_RB_비전이상 AT %MW84042.14 : BOOL;
    R101_1_1_I_RB_실러이상 AT %MW84042.13 : BOOL;
    R101_1_1_I_RB_용접카운터이상 AT %MW84042.15 : BOOL;
    R101_1_1_I_RB_용접타점수 AT %MW84045 : WORD;
    R101_1_1_I_RB_운전준비 AT %MW84040.3 : BOOL;
    R101_1_1_I_RB_원위치 AT %MW84040.0 : BOOL;
    R101_1_1_I_RB_이상리셋 AT %MW84040.2 : BOOL;
    R101_1_1_I_RB_자동 AT %MW84040.4 : BOOL;
    R101_1_1_I_RB_자동기동 AT %MW84040.5 : BOOL;
    R101_1_1_I_RB_최종_작업완료 AT %MW84040.1 : BOOL;
    R101_1_1_I_RB_통신이상 AT %MW84042.12 : BOOL;
    R101_1_1_M_DATA_삭제_PLS AT %MW9000.0 : BOOL; (* R101_1_1_M_DATA_삭제_PLS *)
    R101_1_1_M_DATA_삭제_SIGN AT %MW9000.1 : BOOL; (* R101_1_1_M_DATA_삭제_SIGN *)
    R101_1_1_M_DATA_삭제_완료 AT %MW9000.2 : BOOL; (* R101_1_1_M_DATA_삭제_완료 *)
    R101_1_1_M_DATA_전송_MEMO AT %MW9000.8 : BOOL; (* R101_1_1_M_DATA_전송_MEMO *)
    R101_1_1_M_DATA_전송_PLS AT %MW9000.9 : BOOL; (* R101_1_1_M_DATA_전송_PLS *)
    R101_1_1_M_DATA_전송_SIGN AT %MW9000.10 : BOOL; (* R101_1_1_M_DATA_전송_SIGN *)
    R101_1_1_M_DATA_전송_완료 AT %MW9000.11 : BOOL; (* R101_1_1_M_DATA_전송_완료 *)
    R101_1_1_M_I_RB_1차_작업완료 AT %MW20041.2 : BOOL;
    R101_1_1_M_I_RB_2차_작업완료 AT %MW20041.3 : BOOL;
    R101_1_1_M_I_RB_3차_작업완료 AT %MW20041.4 : BOOL;
    R101_1_1_M_I_RB_4차_작업완료 AT %MW20041.5 : BOOL;
    R101_1_1_M_I_RB_5차_작업완료 AT %MW20041.6 : BOOL;
    R101_1_1_M_I_RB_6차_작업완료 AT %MW20041.7 : BOOL;
    R101_1_1_M_I_RB_7차_작업완료 AT %MW20041.8 : BOOL;
    R101_1_1_M_I_RB_PAUSE_보조 AT %MW20040.5 : BOOL;
    R101_1_1_M_I_RB_PLC_RUN_CHK_이상 AT %MW20040.7 : BOOL;
    R101_1_1_M_I_RB_간섭무_1 AT %MW20042.0 : BOOL;
    R101_1_1_M_I_RB_간섭무_10 AT %MW20042.9 : BOOL;
    R101_1_1_M_I_RB_간섭무_11 AT %MW20042.10 : BOOL;
    R101_1_1_M_I_RB_간섭무_12 AT %MW20042.11 : BOOL;
    R101_1_1_M_I_RB_간섭무_2 AT %MW20042.1 : BOOL;
    R101_1_1_M_I_RB_간섭무_3 AT %MW20042.2 : BOOL;
    R101_1_1_M_I_RB_간섭무_4 AT %MW20042.3 : BOOL;
    R101_1_1_M_I_RB_간섭무_5 AT %MW20042.4 : BOOL;
    R101_1_1_M_I_RB_간섭무_6 AT %MW20042.5 : BOOL;
    R101_1_1_M_I_RB_간섭무_7 AT %MW20042.6 : BOOL;
    R101_1_1_M_I_RB_간섭무_8 AT %MW20042.7 : BOOL;
    R101_1_1_M_I_RB_간섭무_9 AT %MW20042.8 : BOOL;
    R101_1_1_M_I_RB_비상정지 AT %MW20040.4 : BOOL;
    R101_1_1_M_I_RB_운전준비 AT %MW20040.0 : BOOL;
    R101_1_1_M_I_RB_원위치 AT %MW20040.3 : BOOL;
    R101_1_1_M_I_RB_이상 AT %MW20040.2 : BOOL;
    R101_1_1_M_I_RB_자동 AT %MW20040.1 : BOOL;
    R101_1_1_M_I_RB_최종작업완료 AT %MW20041.0 : BOOL;
    R101_1_1_M_I_RB_프로그램_이상 AT %MW20040.6 : BOOL;
    R101_1_1_M_O_RB_1_CYCLE_SET AT %MW21040.3 : BOOL;
    R101_1_1_M_O_RB_1_CYCLE_리셋 AT %MW21040.4 : BOOL;
    R101_1_1_M_O_RB_1차_작업완료_리셋 AT %MW21042.0 : BOOL;
    R101_1_1_M_O_RB_2차_작업완료_리셋 AT %MW21042.1 : BOOL;
    R101_1_1_M_O_RB_2차_진입OK AT %MW21041.8 : BOOL;
    R101_1_1_M_O_RB_3차_작업완료_리셋 AT %MW21042.2 : BOOL;
    R101_1_1_M_O_RB_3차_진입OK AT %MW21041.9 : BOOL;
    R101_1_1_M_O_RB_4차_작업완료_리셋 AT %MW21042.3 : BOOL;
    R101_1_1_M_O_RB_4차_진입OK AT %MW21041.10 : BOOL;
    R101_1_1_M_O_RB_5차_작업완료_리셋 AT %MW21042.4 : BOOL;
    R101_1_1_M_O_RB_5차_진입OK AT %MW21041.11 : BOOL;
    R101_1_1_M_O_RB_6차_작업완료_리셋 AT %MW21042.5 : BOOL;
    R101_1_1_M_O_RB_6차_진입OK AT %MW21041.12 : BOOL;
    R101_1_1_M_O_RB_7차_작업완료_리셋 AT %MW21042.6 : BOOL;
    R101_1_1_M_O_RB_7차_진입OK AT %MW21041.13 : BOOL;
    R101_1_1_M_O_RB_ATD_OK AT %MW21040.6 : BOOL;
    R101_1_1_M_O_RB_PLT_10_진입OK AT %MW21043.10 : BOOL;
    R101_1_1_M_O_RB_PLT_11_진입OK AT %MW21043.11 : BOOL;
    R101_1_1_M_O_RB_PLT_12_진입OK AT %MW21043.12 : BOOL;
    R101_1_1_M_O_RB_PLT_1_진입OK AT %MW21043.1 : BOOL;
    R101_1_1_M_O_RB_PLT_2_진입OK AT %MW21043.2 : BOOL;
    R101_1_1_M_O_RB_PLT_3_진입OK AT %MW21043.3 : BOOL;
    R101_1_1_M_O_RB_PLT_4_진입OK AT %MW21043.4 : BOOL;
    R101_1_1_M_O_RB_PLT_5_진입OK AT %MW21043.5 : BOOL;
    R101_1_1_M_O_RB_PLT_6_진입OK AT %MW21043.6 : BOOL;
    R101_1_1_M_O_RB_PLT_7_진입OK AT %MW21043.7 : BOOL;
    R101_1_1_M_O_RB_PLT_8_진입OK AT %MW21043.8 : BOOL;
    R101_1_1_M_O_RB_PLT_9_진입OK AT %MW21043.9 : BOOL;
    R101_1_1_M_O_RB_PLT_카운터리셋_보조 AT %MW21040.10 : BOOL;
    R101_1_1_M_O_RB_RESTART_OK AT %MW21040.2 : BOOL;
    R101_1_1_M_O_RB_START_OK AT %MW21040.0 : BOOL;
    R101_1_1_M_O_RB_TEST_MODE_5000회 AT %MW21040.12 : BOOL;
    R101_1_1_M_O_RB_TIP_교체_시작 AT %MW21040.7 : BOOL;
    R101_1_1_M_O_RB_TIP_교체_완료 AT %MW21040.8 : BOOL;
    R101_1_1_M_O_RB_VIP_MODE AT %MW21040.11 : BOOL;
    R101_1_1_M_O_RB_냉각수_차단_요청 AT %MW21040.9 : BOOL;
    R101_1_1_M_O_RB_진입OK_AX차종 AT %MW21041.0 : BOOL;
    R101_1_1_M_O_RB_진입OK_B차종 AT %MW21041.1 : BOOL;
    R101_1_1_M_O_RB_진입OK_C차종 AT %MW21041.2 : BOOL;
    R101_1_1_M_O_RB_진입OK_D차종 AT %MW21041.3 : BOOL;
    R101_1_1_M_O_RB_진입OK_E차종 AT %MW21041.4 : BOOL;
    R101_1_1_M_O_RB_진입OK_F차종 AT %MW21041.5 : BOOL;
    R101_1_1_M_O_RB_진입OK_G차종 AT %MW21041.6 : BOOL;
    R101_1_1_M_O_RB_진입OK_H차종 AT %MW21041.7 : BOOL;
    R101_1_1_M_O_RB_최종_작업완료_리셋 AT %MW21040.5 : BOOL;
    R101_1_1_M_O_RB_프로그램_OK AT %MW21040.1 : BOOL;
    R101_1_1_M_RB_PROG_NO AT %MW20044 : WORD;
    R101_1_1_M_RB_통신이상 AT %MW1024.10 : BOOL;
    R101_1_1_M_SEQ AT %MW10000 : WORD; (* R101_1_1_M_SEQ *)
    R101_1_1_M_STN_차종_NONE AT %MW1002.3 : BOOL;
    R101_1_1_M_STN_차종_ON AT %MW1002.2 : BOOL;
    R101_1_1_M_VIN_NO_1_2 AT %MW10011 : WORD; (* R101_1_1_M_VIN_NO_1_2 *)
    R101_1_1_M_VIN_NO_3_4 AT %MW10012 : WORD; (* R101_1_1_M_VIN_NO_3_4 *)
    R101_1_1_M_VIN_NO_5_6 AT %MW10013 : WORD; (* R101_1_1_M_VIN_NO_5_6 *)
    R101_1_1_M_VIN_NO_7_8 AT %MW10014 : WORD; (* R101_1_1_M_VIN_NO_7_8 *)
    R101_1_1_M_VIN_NO_9_10 AT %MW10015 : WORD; (* R101_1_1_M_VIN_NO_9_10 *)
    R101_1_1_M_차종1_AX AT %MW10001.0 : BOOL; (* R101_1_1_M_차종1_AX *)
    R101_1_1_M_차종1_B AT %MW10001.1 : BOOL; (* R101_1_1_M_차종1_B *)
    R101_1_1_M_차종1_C AT %MW10001.2 : BOOL; (* R101_1_1_M_차종1_C *)
    R101_1_1_M_차종1_D AT %MW10001.3 : BOOL; (* R101_1_1_M_차종1_D *)
    R101_1_1_M_차종1_E AT %MW10001.4 : BOOL; (* R101_1_1_M_차종1_E *)
    R101_1_1_M_차종1_F AT %MW10001.5 : BOOL; (* R101_1_1_M_차종1_F *)
    R101_1_1_M_차종1_G AT %MW10001.6 : BOOL; (* R101_1_1_M_차종1_G *)
    R101_1_1_M_차종1_H AT %MW10001.7 : BOOL; (* R101_1_1_M_차종1_H *)
    R101_1_1_M_차종2_3DR AT %MW10001.8 : BOOL; (* R101_1_1_M_차종2_3DR *)
    R101_1_1_M_차종2_4DR AT %MW10001.9 : BOOL; (* R101_1_1_M_차종2_4DR *)
    R101_1_1_M_차종2_5DR AT %MW10001.10 : BOOL; (* R101_1_1_M_차종2_5DR *)
    R101_1_1_M_차종2_SP1 AT %MW10001.12 : BOOL; (* R101_1_1_M_차종2_SP1 *)
    R101_1_1_M_차종2_SP2 AT %MW10001.13 : BOOL; (* R101_1_1_M_차종2_SP2 *)
    R101_1_1_M_차종2_WGN AT %MW10001.11 : BOOL; (* R101_1_1_M_차종2_WGN *)
    R101_1_1_M_차종3_LHD AT %MW10001.14 : BOOL; (* R101_1_1_M_차종3_LHD *)
    R101_1_1_M_차종3_RHD AT %MW10001.15 : BOOL; (* R101_1_1_M_차종3_RHD *)
    R101_1_1_M_차종4_EEC AT %MW10002.3 : BOOL; (* R101_1_1_M_차종4_EEC *)
    R101_1_1_M_차종4_SP1 AT %MW10002.8 : BOOL; (* R101_1_1_M_차종4_SP1 *)
    R101_1_1_M_차종4_SP2 AT %MW10002.9 : BOOL; (* R101_1_1_M_차종4_SP2 *)
    R101_1_1_M_차종4_SP3 AT %MW10002.11 : BOOL; (* R101_1_1_M_차종4_SP3 *)
    R101_1_1_M_차종4_SP4 AT %MW10002.12 : BOOL; (* R101_1_1_M_차종4_SP4 *)
    R101_1_1_M_차종4_SP5 AT %MW10002.13 : BOOL; (* R101_1_1_M_차종4_SP5 *)
    R101_1_1_M_차종4_SP6 AT %MW10002.14 : BOOL; (* R101_1_1_M_차종4_SP6 *)
    R101_1_1_M_차종4_SP7 AT %MW10002.15 : BOOL; (* R101_1_1_M_차종4_SP7 *)
    R101_1_1_M_차종4_내수 AT %MW10002.0 : BOOL; (* R101_1_1_M_차종4_내수 *)
    R101_1_1_M_차종4_러시아 AT %MW10002.10 : BOOL; (* R101_1_1_M_차종4_러시아 *)
    R101_1_1_M_차종4_북미 AT %MW10002.2 : BOOL; (* R101_1_1_M_차종4_북미 *)
    R101_1_1_M_차종4_브라질 AT %MW10002.7 : BOOL; (* R101_1_1_M_차종4_브라질 *)
    R101_1_1_M_차종4_수출 AT %MW10002.1 : BOOL; (* R101_1_1_M_차종4_수출 *)
    R101_1_1_M_차종4_중국 AT %MW10002.6 : BOOL; (* R101_1_1_M_차종4_중국 *)
    R101_1_1_M_차종4_중동 AT %MW10002.5 : BOOL; (* R101_1_1_M_차종4_중동 *)
    R101_1_1_M_차종4_호주 AT %MW10002.4 : BOOL; (* R101_1_1_M_차종4_호주 *)
    R101_1_1_M_차종5_AT AT %MW10003.1 : BOOL; (* R101_1_1_M_차종5_AT *)
    R101_1_1_M_차종5_MT AT %MW10003.0 : BOOL; (* R101_1_1_M_차종5_MT *)
    R101_1_1_M_차종5_SP1 AT %MW10003.2 : BOOL; (* R101_1_1_M_차종5_SP1 *)
    R101_1_1_M_차종6_DSROOF AT %MW10003.6 : BOOL; (* R101_1_1_M_차종6_DSROOF *)
    R101_1_1_M_차종6_SP1 AT %MW10003.7 : BOOL; (* R101_1_1_M_차종6_SP1 *)
    R101_1_1_M_차종6_썬루프 AT %MW10003.4 : BOOL; (* R101_1_1_M_차종6_썬루프 *)
    R101_1_1_M_차종6_일반루프 AT %MW10003.3 : BOOL; (* R101_1_1_M_차종6_일반루프 *)
    R101_1_1_M_차종6_파노라마루프 AT %MW10003.5 : BOOL; (* R101_1_1_M_차종6_파노라마루프 *)
    R101_1_1_M_차종7_DSL AT %MW10003.9 : BOOL; (* R101_1_1_M_차종7_DSL *)
    R101_1_1_M_차종7_GSL AT %MW10003.8 : BOOL; (* R101_1_1_M_차종7_GSL *)
    R101_1_1_M_차종7_SP1 AT %MW10003.10 : BOOL; (* R101_1_1_M_차종7_SP1 *)
    R101_1_1_M_차종7_SP2 AT %MW10003.11 : BOOL; (* R101_1_1_M_차종7_SP2 *)
    R101_1_1_M_차종7_SP3 AT %MW10003.12 : BOOL; (* R101_1_1_M_차종7_SP3 *)
    R101_1_1_M_차종7_SP4 AT %MW10003.13 : BOOL; (* R101_1_1_M_차종7_SP4 *)
    R101_1_1_M_차종7_SP5 AT %MW10003.14 : BOOL; (* R101_1_1_M_차종7_SP5 *)
    R101_1_1_M_차종7_SP6 AT %MW10003.15 : BOOL; (* R101_1_1_M_차종7_SP6 *)
    R101_1_1_M_차종8_2WD AT %MW10004.0 : BOOL; (* R101_1_1_M_차종8_2WD *)
    R101_1_1_M_차종8_4WD AT %MW10004.1 : BOOL; (* R101_1_1_M_차종8_4WD *)
    R101_1_1_M_차종8_SP1 AT %MW10004.2 : BOOL; (* R101_1_1_M_차종8_SP1 *)
    R101_1_1_M_차종9_MPI AT %MW10004.3 : BOOL; (* R101_1_1_M_차종9_MPI *)
    R101_1_1_M_차종9_SP1 AT %MW10004.5 : BOOL; (* R101_1_1_M_차종9_SP1 *)
    R101_1_1_M_차종9_SP10 AT %MW10004.14 : BOOL; (* R101_1_1_M_차종9_SP10 *)
    R101_1_1_M_차종9_SP11 AT %MW10004.15 : BOOL; (* R101_1_1_M_차종9_SP11 *)
    R101_1_1_M_차종9_SP2 AT %MW10004.6 : BOOL; (* R101_1_1_M_차종9_SP2 *)
    R101_1_1_M_차종9_SP3 AT %MW10004.7 : BOOL; (* R101_1_1_M_차종9_SP3 *)
    R101_1_1_M_차종9_SP4 AT %MW10004.8 : BOOL; (* R101_1_1_M_차종9_SP4 *)
    R101_1_1_M_차종9_SP5 AT %MW10004.9 : BOOL; (* R101_1_1_M_차종9_SP5 *)
    R101_1_1_M_차종9_SP6 AT %MW10004.10 : BOOL; (* R101_1_1_M_차종9_SP6 *)
    R101_1_1_M_차종9_SP7 AT %MW10004.11 : BOOL; (* R101_1_1_M_차종9_SP7 *)
    R101_1_1_M_차종9_SP8 AT %MW10004.12 : BOOL; (* R101_1_1_M_차종9_SP8 *)
    R101_1_1_M_차종9_SP9 AT %MW10004.13 : BOOL; (* R101_1_1_M_차종9_SP9 *)
    R101_1_1_M_차종9_T_GDI AT %MW10004.4 : BOOL; (* R101_1_1_M_차종9_T_GDI *)
    R101_1_1_M_차종_AS AT %MW10010.9 : BOOL; (* R101_1_1_M_차종_AS *)
    R101_1_1_M_차종_OPT1_R_RACK_무 AT %MW10005.3 : BOOL; (* R101_1_1_M_차종_OPT1_R_RACK_무 *)
    R101_1_1_M_차종_OPT1_R_RACK_유 AT %MW10005.2 : BOOL; (* R101_1_1_M_차종_OPT1_R_RACK_유 *)
    R101_1_1_M_차종_OPT1_SP1 AT %MW10005.10 : BOOL; (* R101_1_1_M_차종_OPT1_SP1 *)
    R101_1_1_M_차종_OPT1_SP2 AT %MW10005.11 : BOOL; (* R101_1_1_M_차종_OPT1_SP2 *)
    R101_1_1_M_차종_OPT1_SP3 AT %MW10005.12 : BOOL; (* R101_1_1_M_차종_OPT1_SP3 *)
    R101_1_1_M_차종_OPT1_SP4 AT %MW10005.13 : BOOL; (* R101_1_1_M_차종_OPT1_SP4 *)
    R101_1_1_M_차종_OPT1_SP5 AT %MW10005.14 : BOOL; (* R101_1_1_M_차종_OPT1_SP5 *)
    R101_1_1_M_차종_OPT1_SP6 AT %MW10005.15 : BOOL; (* R101_1_1_M_차종_OPT1_SP6 *)
    R101_1_1_M_차종_OPT1_S_REP_EATER_무 AT %MW10005.7 : BOOL; (* R101_1_1_M_차종_OPT1_S_REP_EATER_무 *)
    R101_1_1_M_차종_OPT1_S_REP_EATER_유 AT %MW10005.6 : BOOL; (* R101_1_1_M_차종_OPT1_S_REP_EATER_유 *)
    R101_1_1_M_차종_OPT1_VAN_무 AT %MW10005.9 : BOOL; (* R101_1_1_M_차종_OPT1_VAN_무 *)
    R101_1_1_M_차종_OPT1_VAN_유 AT %MW10005.8 : BOOL; (* R101_1_1_M_차종_OPT1_VAN_유 *)
    R101_1_1_M_차종_OPT1_슬라이딩_무 AT %MW10005.1 : BOOL; (* R101_1_1_M_차종_OPT1_슬라이딩_무 *)
    R101_1_1_M_차종_OPT1_슬라이딩_유 AT %MW10005.0 : BOOL; (* R101_1_1_M_차종_OPT1_슬라이딩_유 *)
    R101_1_1_M_차종_OPT1_폴딩_무 AT %MW10005.5 : BOOL; (* R101_1_1_M_차종_OPT1_폴딩_무 *)
    R101_1_1_M_차종_OPT1_폴딩_유 AT %MW10005.4 : BOOL; (* R101_1_1_M_차종_OPT1_폴딩_유 *)
    R101_1_1_M_차종_OPT2_SP_WORD1 AT %MW10006 : WORD; (* R101_1_1_M_차종_OPT2_SP_WORD1 *)
    R101_1_1_M_차종_OPT3_SP_WORD2 AT %MW10007 : WORD; (* R101_1_1_M_차종_OPT3_SP_WORD2 *)
    R101_1_1_M_차종_OPT4_SP_WORD3 AT %MW10008 : WORD; (* R101_1_1_M_차종_OPT4_SP_WORD3 *)
    R101_1_1_M_차종_OPT5_SP_WORD4 AT %MW10009 : WORD; (* R101_1_1_M_차종_OPT5_SP_WORD4 *)
    R101_1_1_M_차종_SP1 AT %MW10010.0 : BOOL; (* R101_1_1_M_차종_SP1 *)
    R101_1_1_M_차종_SP2 AT %MW10010.1 : BOOL; (* R101_1_1_M_차종_SP2 *)
    R101_1_1_M_차종_SP3 AT %MW10010.2 : BOOL; (* R101_1_1_M_차종_SP3 *)
    R101_1_1_M_차종_SP4 AT %MW10010.3 : BOOL; (* R101_1_1_M_차종_SP4 *)
    R101_1_1_M_차종_SP5 AT %MW10010.4 : BOOL; (* R101_1_1_M_차종_SP5 *)
    R101_1_1_M_차종_SP6 AT %MW10010.5 : BOOL; (* R101_1_1_M_차종_SP6 *)
    R101_1_1_M_차종_SP7 AT %MW10010.6 : BOOL; (* R101_1_1_M_차종_SP7 *)
    R101_1_1_M_차종_SP8 AT %MW10010.7 : BOOL; (* R101_1_1_M_차종_SP8 *)
    R101_1_1_M_차종_SP9 AT %MW10010.15 : BOOL; (* R101_1_1_M_차종_SP9 *)
    R101_1_1_M_차종_공대차 AT %MW10010.12 : BOOL; (* R101_1_1_M_차종_공대차 *)
    R101_1_1_M_차종_공차 AT %MW10010.10 : BOOL; (* R101_1_1_M_차종_공차 *)
    R101_1_1_M_차종_불량대차 AT %MW10010.13 : BOOL; (* R101_1_1_M_차종_불량대차 *)
    R101_1_1_M_차종_불량차 AT %MW10010.11 : BOOL; (* R101_1_1_M_차종_불량차 *)
    R101_1_1_M_차종_비축 AT %MW10010.8 : BOOL; (* R101_1_1_M_차종_비축 *)
    R101_1_1_M_차종_취출대차 AT %MW10010.14 : BOOL; (* R101_1_1_M_차종_취출대차 *)
    R101_1_1_O_RB_0_5S_통신_CHK AT %MW94043.14 : BOOL;
    R101_1_1_O_RB_2차_진입OK AT %MW94041.8 : BOOL;
    R101_1_1_O_RB_3차_진입OK AT %MW94041.9 : BOOL;
    R101_1_1_O_RB_4차_진입OK AT %MW94041.10 : BOOL;
    R101_1_1_O_RB_5차_진입OK AT %MW94041.11 : BOOL;
    R101_1_1_O_RB_6차_진입OK AT %MW94041.12 : BOOL;
    R101_1_1_O_RB_7차_진입OK AT %MW94041.13 : BOOL;
    R101_1_1_O_RB_AX_1차_진입OK AT %MW94041.0 : BOOL;
    R101_1_1_O_RB_B_1차_진입OK AT %MW94041.1 : BOOL;
    R101_1_1_O_RB_C_1차_진입OK AT %MW94041.2 : BOOL;
    R101_1_1_O_RB_D_1차_진입OK AT %MW94041.3 : BOOL;
    R101_1_1_O_RB_EACH_작업완료_리셋 AT %MW94040.14 : BOOL;
    R101_1_1_O_RB_EXT_READY AT %MW94040.11 : BOOL;
    R101_1_1_O_RB_E_1차_진입OK AT %MW94041.4 : BOOL;
    R101_1_1_O_RB_F_1차_진입OK AT %MW94041.5 : BOOL;
    R101_1_1_O_RB_GATE_OPEN_NC AT %MW94043.11 : BOOL;
    R101_1_1_O_RB_G_1차_진입OK AT %MW94041.6 : BOOL;
    R101_1_1_O_RB_H_1차_진입OK AT %MW94041.7 : BOOL;
    R101_1_1_O_RB_MUTUAL_INT1 AT %MW94043.0 : BOOL;
    R101_1_1_O_RB_MUTUAL_INT2 AT %MW94043.1 : BOOL;
    R101_1_1_O_RB_MUTUAL_INT3 AT %MW94043.2 : BOOL;
    R101_1_1_O_RB_MUTUAL_INT4 AT %MW94043.3 : BOOL;
    R101_1_1_O_RB_MUTUAL_INT5 AT %MW94043.4 : BOOL;
    R101_1_1_O_RB_MUTUAL_INT6 AT %MW94043.5 : BOOL;
    R101_1_1_O_RB_MUTUAL_INT7 AT %MW94043.6 : BOOL;
    R101_1_1_O_RB_MUTUAL_INT8 AT %MW94043.7 : BOOL;
    R101_1_1_O_RB_OUTPUT AT %MW94040 : ARRAY[0..3] OF WORD;
    R101_1_1_O_RB_PAUSE_NC AT %MW94040.13 : BOOL;
    R101_1_1_O_RB_PLT10_진입OK AT %MW94042.9 : BOOL;
    R101_1_1_O_RB_PLT11_진입OK AT %MW94042.10 : BOOL;
    R101_1_1_O_RB_PLT12_진입OK AT %MW94042.11 : BOOL;
    R101_1_1_O_RB_PLT1_진입OK AT %MW94042.0 : BOOL;
    R101_1_1_O_RB_PLT2_진입OK AT %MW94042.1 : BOOL;
    R101_1_1_O_RB_PLT3_진입OK AT %MW94042.2 : BOOL;
    R101_1_1_O_RB_PLT4_진입OK AT %MW94042.3 : BOOL;
    R101_1_1_O_RB_PLT5_진입OK AT %MW94042.4 : BOOL;
    R101_1_1_O_RB_PLT6_진입OK AT %MW94042.5 : BOOL;
    R101_1_1_O_RB_PLT7_진입OK AT %MW94042.6 : BOOL;
    R101_1_1_O_RB_PLT8_진입OK AT %MW94042.7 : BOOL;
    R101_1_1_O_RB_PLT9_진입OK AT %MW94042.8 : BOOL;
    R101_1_1_O_RB_PLT_COUNT_리셋_COND AT %MW94043.10 : BOOL;
    R101_1_1_O_RB_PROG_선택1 AT %MW94040.0 : BOOL;
    R101_1_1_O_RB_PROG_선택128 AT %MW94040.7 : BOOL;
    R101_1_1_O_RB_PROG_선택16 AT %MW94040.4 : BOOL;
    R101_1_1_O_RB_PROG_선택2 AT %MW94040.1 : BOOL;
    R101_1_1_O_RB_PROG_선택32 AT %MW94040.5 : BOOL;
    R101_1_1_O_RB_PROG_선택4 AT %MW94040.2 : BOOL;
    R101_1_1_O_RB_PROG_선택64 AT %MW94040.6 : BOOL;
    R101_1_1_O_RB_PROG_선택8 AT %MW94040.3 : BOOL;
    R101_1_1_O_RB_SP_1_14 AT %MW94041.14 : BOOL;
    R101_1_1_O_RB_SP_1_15 AT %MW94041.15 : BOOL;
    R101_1_1_O_RB_SP_2_12 AT %MW94042.12 : BOOL;
    R101_1_1_O_RB_SP_2_13 AT %MW94042.13 : BOOL;
    R101_1_1_O_RB_SP_2_14 AT %MW94042.14 : BOOL;
    R101_1_1_O_RB_SP_5000TH_ON AT %MW94042.15 : BOOL;
    R101_1_1_O_RB_TIP_CHANGE_END AT %MW94043.9 : BOOL;
    R101_1_1_O_RB_TIP_CHANGE_START AT %MW94043.8 : BOOL;
    R101_1_1_O_RB_TIP_DRESS_SATRT AT %MW94040.12 : BOOL;
    R101_1_1_O_RB_VIP_MODE AT %MW94043.15 : BOOL;
    R101_1_1_O_RB_기동 AT %MW94040.9 : BOOL;
    R101_1_1_O_RB_냉각수차단 AT %MW94040.15 : BOOL;
    R101_1_1_O_RB_부저정지 AT %MW94043.13 : BOOL;
    R101_1_1_O_RB_비상정지_NC AT %MW94043.12 : BOOL;
    R101_1_1_O_RB_이상_리셋 AT %MW94040.10 : BOOL;
    R101_1_1_O_RB_작업완료_리셋 AT %MW94040.8 : BOOL;
    R101_1_I_RB_0_5_COMM_CHK AT %MW84073.14 : BOOL;
    R101_1_I_RB_10차_간섭무 AT %MW84071.9 : BOOL;
    R101_1_I_RB_11차_간섭무 AT %MW84071.10 : BOOL;
    R101_1_I_RB_12차_간섭무 AT %MW84071.11 : BOOL;
    R101_1_I_RB_1차_간섭무 AT %MW84071.0 : BOOL;
    R101_1_I_RB_1차_작업완료 AT %MW84070.9 : BOOL;
    R101_1_I_RB_2차_간섭무 AT %MW84071.1 : BOOL;
    R101_1_I_RB_2차_작업완료 AT %MW84070.10 : BOOL;
    R101_1_I_RB_3차_간섭무 AT %MW84071.2 : BOOL;
    R101_1_I_RB_3차_작업완료 AT %MW84070.11 : BOOL;
    R101_1_I_RB_4차_간섭무 AT %MW84071.3 : BOOL;
    R101_1_I_RB_4차_작업완료 AT %MW84070.12 : BOOL;
    R101_1_I_RB_5차_간섭무 AT %MW84071.4 : BOOL;
    R101_1_I_RB_5차_작업완료 AT %MW84070.13 : BOOL;
    R101_1_I_RB_6차_간섭무 AT %MW84071.5 : BOOL;
    R101_1_I_RB_6차_작업완료 AT %MW84070.14 : BOOL;
    R101_1_I_RB_7차_간섭무 AT %MW84071.6 : BOOL;
    R101_1_I_RB_7차_작업완료 AT %MW84070.15 : BOOL;
    R101_1_I_RB_8차_간섭무 AT %MW84071.7 : BOOL;
    R101_1_I_RB_9차_간섭무 AT %MW84071.8 : BOOL;
    R101_1_I_RB_AB_NORMAL_선택 AT %MW84070.6 : BOOL;
    R101_1_I_RB_GUN1_FIXED_TIP AT %MW84077 : WORD;
    R101_1_I_RB_GUN1_MOVING_TIP AT %MW84076 : WORD;
    R101_1_I_RB_GUN2_FIXED_TIP AT %MW84079 : WORD;
    R101_1_I_RB_GUN2_MOVING_TIP AT %MW84078 : WORD;
    R101_1_I_RB_INPUT AT %MW84070 : ARRAY[0..3] OF WORD;
    R101_1_I_RB_LS_이상 AT %MW84072.11 : BOOL;
    R101_1_I_RB_MOTOR_MC_ON AT %MW84073.15 : BOOL;
    R101_1_I_RB_MUTUAL_INT1 AT %MW84073.0 : BOOL;
    R101_1_I_RB_MUTUAL_INT2 AT %MW84073.1 : BOOL;
    R101_1_I_RB_MUTUAL_INT3 AT %MW84073.2 : BOOL;
    R101_1_I_RB_MUTUAL_INT4 AT %MW84073.3 : BOOL;
    R101_1_I_RB_MUTUAL_INT5 AT %MW84073.4 : BOOL;
    R101_1_I_RB_MUTUAL_INT6 AT %MW84073.5 : BOOL;
    R101_1_I_RB_MUTUAL_INT7 AT %MW84073.6 : BOOL;
    R101_1_I_RB_MUTUAL_INT8 AT %MW84073.7 : BOOL;
    R101_1_I_RB_PLT_UNLOAD_완료 AT %MW84073.11 : BOOL;
    R101_1_I_RB_PLT_최종UNLOAD_완료 AT %MW84073.12 : BOOL;
    R101_1_I_RB_PROG_ECHO_1 AT %MW84072.0 : BOOL;
    R101_1_I_RB_PROG_ECHO_128 AT %MW84072.7 : BOOL;
    R101_1_I_RB_PROG_ECHO_16 AT %MW84072.4 : BOOL;
    R101_1_I_RB_PROG_ECHO_2 AT %MW84072.1 : BOOL;
    R101_1_I_RB_PROG_ECHO_32 AT %MW84072.5 : BOOL;
    R101_1_I_RB_PROG_ECHO_4 AT %MW84072.2 : BOOL;
    R101_1_I_RB_PROG_ECHO_64 AT %MW84072.6 : BOOL;
    R101_1_I_RB_PROG_ECHO_8 AT %MW84072.3 : BOOL;
    R101_1_I_RB_SP3_8 AT %MW84073.8 : BOOL;
    R101_1_I_RB_SP3_9 AT %MW84073.9 : BOOL;
    R101_1_I_RB_SPARE_WORD_4 AT %MW84074 : WORD;
    R101_1_I_RB_SP_1_12 AT %MW84071.12 : BOOL;
    R101_1_I_RB_SP_1_13 AT %MW84071.13 : BOOL;
    R101_1_I_RB_SP_1_14 AT %MW84071.14 : BOOL;
    R101_1_I_RB_SP_1_15 AT %MW84071.15 : BOOL;
    R101_1_I_RB_TC_이상 AT %MW84072.8 : BOOL;
    R101_1_I_RB_TIP_CHANGE AT %MW84073.13 : BOOL;
    R101_1_I_RB_TIP_DRESSING AT %MW84070.7 : BOOL;
    R101_1_I_RB__PLT_카운터리셋완료 AT %MW84073.10 : BOOL;
    R101_1_I_RB_공기압_이상 AT %MW84072.9 : BOOL;
    R101_1_I_RB_냉각수_이상 AT %MW84072.10 : BOOL;
    R101_1_I_RB_비상정지_NC AT %MW84070.8 : BOOL;
    R101_1_I_RB_비전이상 AT %MW84072.14 : BOOL;
    R101_1_I_RB_실러이상 AT %MW84072.13 : BOOL;
    R101_1_I_RB_용접카운터이상 AT %MW84072.15 : BOOL;
    R101_1_I_RB_용접타점수 AT %MW84075 : WORD;
    R101_1_I_RB_운전준비 AT %MW84070.3 : BOOL;
    R101_1_I_RB_원위치 AT %MW84070.0 : BOOL;
    R101_1_I_RB_이상리셋 AT %MW84070.2 : BOOL;
    R101_1_I_RB_자동 AT %MW84070.4 : BOOL;
    R101_1_I_RB_자동기동 AT %MW84070.5 : BOOL;
    R101_1_I_RB_최종_작업완료 AT %MW84070.1 : BOOL;
    R101_1_I_RB_통신이상 AT %MW84072.12 : BOOL;
    R101_1_M_AX_차종_용접타점수 AT %MW8110 : WORD; (* R101_1_M_AX_차종_용접타점수 *)
    R101_1_M_I_RB_1차_작업완료 AT %MW20071.2 : BOOL;
    R101_1_M_I_RB_2차_작업완료 AT %MW20071.3 : BOOL;
    R101_1_M_I_RB_3차_작업완료 AT %MW20071.4 : BOOL;
    R101_1_M_I_RB_4차_작업완료 AT %MW20071.5 : BOOL;
    R101_1_M_I_RB_5차_작업완료 AT %MW20071.6 : BOOL;
    R101_1_M_I_RB_6차_작업완료 AT %MW20071.7 : BOOL;
    R101_1_M_I_RB_7차_작업완료 AT %MW20071.8 : BOOL;
    R101_1_M_I_RB_PAUSE_보조 AT %MW20070.5 : BOOL;
    R101_1_M_I_RB_PLC_RUN_CHK_이상 AT %MW20070.7 : BOOL;
    R101_1_M_I_RB_간섭무_1 AT %MW20072.0 : BOOL;
    R101_1_M_I_RB_간섭무_10 AT %MW20072.9 : BOOL;
    R101_1_M_I_RB_간섭무_11 AT %MW20072.10 : BOOL;
    R101_1_M_I_RB_간섭무_12 AT %MW20072.11 : BOOL;
    R101_1_M_I_RB_간섭무_2 AT %MW20072.1 : BOOL;
    R101_1_M_I_RB_간섭무_3 AT %MW20072.2 : BOOL;
    R101_1_M_I_RB_간섭무_4 AT %MW20072.3 : BOOL;
    R101_1_M_I_RB_간섭무_5 AT %MW20072.4 : BOOL;
    R101_1_M_I_RB_간섭무_6 AT %MW20072.5 : BOOL;
    R101_1_M_I_RB_간섭무_7 AT %MW20072.6 : BOOL;
    R101_1_M_I_RB_간섭무_8 AT %MW20072.7 : BOOL;
    R101_1_M_I_RB_간섭무_9 AT %MW20072.8 : BOOL;
    R101_1_M_I_RB_비상정지 AT %MW20070.4 : BOOL;
    R101_1_M_I_RB_운전준비 AT %MW20070.0 : BOOL;
    R101_1_M_I_RB_원위치 AT %MW20070.3 : BOOL;
    R101_1_M_I_RB_이상 AT %MW20070.2 : BOOL;
    R101_1_M_I_RB_자동 AT %MW20070.1 : BOOL;
    R101_1_M_I_RB_최종작업완료 AT %MW20071.0 : BOOL;
    R101_1_M_I_RB_프로그램_이상 AT %MW20070.6 : BOOL;
    R101_1_M_O_RB_1_CYCLE_SET AT %MW21070.3 : BOOL;
    R101_1_M_O_RB_1_CYCLE_리셋 AT %MW21070.4 : BOOL;
    R101_1_M_O_RB_1차_작업완료_리셋 AT %MW21072.0 : BOOL;
    R101_1_M_O_RB_2차_작업완료_리셋 AT %MW21072.1 : BOOL;
    R101_1_M_O_RB_2차_진입OK AT %MW21071.8 : BOOL;
    R101_1_M_O_RB_3차_작업완료_리셋 AT %MW21072.2 : BOOL;
    R101_1_M_O_RB_3차_진입OK AT %MW21071.9 : BOOL;
    R101_1_M_O_RB_4차_작업완료_리셋 AT %MW21072.3 : BOOL;
    R101_1_M_O_RB_4차_진입OK AT %MW21071.10 : BOOL;
    R101_1_M_O_RB_5차_작업완료_리셋 AT %MW21072.4 : BOOL;
    R101_1_M_O_RB_5차_진입OK AT %MW21071.11 : BOOL;
    R101_1_M_O_RB_6차_작업완료_리셋 AT %MW21072.5 : BOOL;
    R101_1_M_O_RB_6차_진입OK AT %MW21071.12 : BOOL;
    R101_1_M_O_RB_7차_작업완료_리셋 AT %MW21072.6 : BOOL;
    R101_1_M_O_RB_7차_진입OK AT %MW21071.13 : BOOL;
    R101_1_M_O_RB_ATD_OK AT %MW21070.6 : BOOL;
    R101_1_M_O_RB_PLT_10_진입OK AT %MW21073.10 : BOOL;
    R101_1_M_O_RB_PLT_11_진입OK AT %MW21073.11 : BOOL;
    R101_1_M_O_RB_PLT_12_진입OK AT %MW21073.12 : BOOL;
    R101_1_M_O_RB_PLT_1_진입OK AT %MW21073.1 : BOOL;
    R101_1_M_O_RB_PLT_2_진입OK AT %MW21073.2 : BOOL;
    R101_1_M_O_RB_PLT_3_진입OK AT %MW21073.3 : BOOL;
    R101_1_M_O_RB_PLT_4_진입OK AT %MW21073.4 : BOOL;
    R101_1_M_O_RB_PLT_5_진입OK AT %MW21073.5 : BOOL;
    R101_1_M_O_RB_PLT_6_진입OK AT %MW21073.6 : BOOL;
    R101_1_M_O_RB_PLT_7_진입OK AT %MW21073.7 : BOOL;
    R101_1_M_O_RB_PLT_8_진입OK AT %MW21073.8 : BOOL;
    R101_1_M_O_RB_PLT_9_진입OK AT %MW21073.9 : BOOL;
    R101_1_M_O_RB_PLT_카운터리셋_보조 AT %MW21070.10 : BOOL;
    R101_1_M_O_RB_RESTART_OK AT %MW21070.2 : BOOL;
    R101_1_M_O_RB_START_OK AT %MW21070.0 : BOOL;
    R101_1_M_O_RB_TEST_MODE_5000회 AT %MW21070.12 : BOOL;
    R101_1_M_O_RB_TIP_교체_시작 AT %MW21070.7 : BOOL;
    R101_1_M_O_RB_TIP_교체_완료 AT %MW21070.8 : BOOL;
    R101_1_M_O_RB_VIP_MODE AT %MW21070.11 : BOOL;
    R101_1_M_O_RB_냉각수_차단_요청 AT %MW21070.9 : BOOL;
    R101_1_M_O_RB_진입OK_AX차종 AT %MW21071.0 : BOOL;
    R101_1_M_O_RB_진입OK_B차종 AT %MW21071.1 : BOOL;
    R101_1_M_O_RB_진입OK_C차종 AT %MW21071.2 : BOOL;
    R101_1_M_O_RB_진입OK_D차종 AT %MW21071.3 : BOOL;
    R101_1_M_O_RB_진입OK_E차종 AT %MW21071.4 : BOOL;
    R101_1_M_O_RB_진입OK_F차종 AT %MW21071.5 : BOOL;
    R101_1_M_O_RB_진입OK_G차종 AT %MW21071.6 : BOOL;
    R101_1_M_O_RB_진입OK_H차종 AT %MW21071.7 : BOOL;
    R101_1_M_O_RB_최종_작업완료_리셋 AT %MW21070.5 : BOOL;
    R101_1_M_O_RB_프로그램_OK AT %MW21070.1 : BOOL;
    R101_1_M_RB_PROG_NO AT %MW20074 : WORD;
    R101_1_M_RB_통신이상 AT %MW1024.11 : BOOL;
    R101_1_M_용접완료 AT %MW1011.1 : BOOL;
    R101_1_M_용접타점수_OK AT %MW1011.5 : BOOL;
    R101_1_M_용접타점수_이상 AT %MW1011.10 : BOOL;
    R101_1_M_차종_MATCH_이상 AT %MW1015.0 : BOOL;
    R101_1_O_RB_0_5S_통신_CHK AT %MW94073.14 : BOOL;
    R101_1_O_RB_2차_진입OK AT %MW94071.8 : BOOL;
    R101_1_O_RB_3차_진입OK AT %MW94071.9 : BOOL;
    R101_1_O_RB_4차_진입OK AT %MW94071.10 : BOOL;
    R101_1_O_RB_5차_진입OK AT %MW94071.11 : BOOL;
    R101_1_O_RB_6차_진입OK AT %MW94071.12 : BOOL;
    R101_1_O_RB_7차_진입OK AT %MW94071.13 : BOOL;
    R101_1_O_RB_AX_1차_진입OK AT %MW94071.0 : BOOL;
    R101_1_O_RB_B_1차_진입OK AT %MW94071.1 : BOOL;
    R101_1_O_RB_C_1차_진입OK AT %MW94071.2 : BOOL;
    R101_1_O_RB_D_1차_진입OK AT %MW94071.3 : BOOL;
    R101_1_O_RB_EACH_작업완료_리셋 AT %MW94070.14 : BOOL;
    R101_1_O_RB_EXT_READY AT %MW94070.11 : BOOL;
    R101_1_O_RB_E_1차_진입OK AT %MW94071.4 : BOOL;
    R101_1_O_RB_F_1차_진입OK AT %MW94071.5 : BOOL;
    R101_1_O_RB_GATE_OPEN_NC AT %MW94073.11 : BOOL;
    R101_1_O_RB_G_1차_진입OK AT %MW94071.6 : BOOL;
    R101_1_O_RB_H_1차_진입OK AT %MW94071.7 : BOOL;
    R101_1_O_RB_MUTUAL_INT1 AT %MW94073.0 : BOOL;
    R101_1_O_RB_MUTUAL_INT2 AT %MW94073.1 : BOOL;
    R101_1_O_RB_MUTUAL_INT3 AT %MW94073.2 : BOOL;
    R101_1_O_RB_MUTUAL_INT4 AT %MW94073.3 : BOOL;
    R101_1_O_RB_MUTUAL_INT5 AT %MW94073.4 : BOOL;
    R101_1_O_RB_MUTUAL_INT6 AT %MW94073.5 : BOOL;
    R101_1_O_RB_MUTUAL_INT7 AT %MW94073.6 : BOOL;
    R101_1_O_RB_MUTUAL_INT8 AT %MW94073.7 : BOOL;
    R101_1_O_RB_OUTPUT AT %MW94070 : ARRAY[0..3] OF WORD;
    R101_1_O_RB_PAUSE_NC AT %MW94070.13 : BOOL;
    R101_1_O_RB_PLT10_진입OK AT %MW94072.9 : BOOL;
    R101_1_O_RB_PLT11_진입OK AT %MW94072.10 : BOOL;
    R101_1_O_RB_PLT12_진입OK AT %MW94072.11 : BOOL;
    R101_1_O_RB_PLT1_진입OK AT %MW94072.0 : BOOL;
    R101_1_O_RB_PLT2_진입OK AT %MW94072.1 : BOOL;
    R101_1_O_RB_PLT3_진입OK AT %MW94072.2 : BOOL;
    R101_1_O_RB_PLT4_진입OK AT %MW94072.3 : BOOL;
    R101_1_O_RB_PLT5_진입OK AT %MW94072.4 : BOOL;
    R101_1_O_RB_PLT6_진입OK AT %MW94072.5 : BOOL;
    R101_1_O_RB_PLT7_진입OK AT %MW94072.6 : BOOL;
    R101_1_O_RB_PLT8_진입OK AT %MW94072.7 : BOOL;
    R101_1_O_RB_PLT9_진입OK AT %MW94072.8 : BOOL;
    R101_1_O_RB_PLT_COUNT_리셋_COND AT %MW94073.10 : BOOL;
    R101_1_O_RB_PROG_선택1 AT %MW94070.0 : BOOL;
    R101_1_O_RB_PROG_선택128 AT %MW94070.7 : BOOL;
    R101_1_O_RB_PROG_선택16 AT %MW94070.4 : BOOL;
    R101_1_O_RB_PROG_선택2 AT %MW94070.1 : BOOL;
    R101_1_O_RB_PROG_선택32 AT %MW94070.5 : BOOL;
    R101_1_O_RB_PROG_선택4 AT %MW94070.2 : BOOL;
    R101_1_O_RB_PROG_선택64 AT %MW94070.6 : BOOL;
    R101_1_O_RB_PROG_선택8 AT %MW94070.3 : BOOL;
    R101_1_O_RB_SP_1_14 AT %MW94071.14 : BOOL;
    R101_1_O_RB_SP_1_15 AT %MW94071.15 : BOOL;
    R101_1_O_RB_SP_2_12 AT %MW94072.12 : BOOL;
    R101_1_O_RB_SP_2_13 AT %MW94072.13 : BOOL;
    R101_1_O_RB_SP_2_14 AT %MW94072.14 : BOOL;
    R101_1_O_RB_SP_5000TH_ON AT %MW94072.15 : BOOL;
    R101_1_O_RB_TIP_CHANGE_END AT %MW94073.9 : BOOL;
    R101_1_O_RB_TIP_CHANGE_START AT %MW94073.8 : BOOL;
    R101_1_O_RB_TIP_DRESS_SATRT AT %MW94070.12 : BOOL;
    R101_1_O_RB_VIP_MODE AT %MW94073.15 : BOOL;
    R101_1_O_RB_기동 AT %MW94070.9 : BOOL;
    R101_1_O_RB_냉각수차단 AT %MW94070.15 : BOOL;
    R101_1_O_RB_부저정지 AT %MW94073.13 : BOOL;
    R101_1_O_RB_비상정지_NC AT %MW94073.12 : BOOL;
    R101_1_O_RB_이상_리셋 AT %MW94070.10 : BOOL;
    R101_1_O_RB_작업완료_리셋 AT %MW94070.8 : BOOL;
    R101_1_S101_CTYPE_MOVE : FB407_Car_Type_Move_Stn_v1;
    R101_1_S102_CTYPE_MOVE : FB407_Car_Type_Move_Stn_v1;
    R101_2_I_RB_0_5_COMM_CHK AT %MW84063.14 : BOOL;
    R101_2_I_RB_10차_간섭무 AT %MW84061.9 : BOOL;
    R101_2_I_RB_11차_간섭무 AT %MW84061.10 : BOOL;
    R101_2_I_RB_12차_간섭무 AT %MW84061.11 : BOOL;
    R101_2_I_RB_1차_간섭무 AT %MW84061.0 : BOOL;
    R101_2_I_RB_1차_작업완료 AT %MW84060.9 : BOOL;
    R101_2_I_RB_2차_간섭무 AT %MW84061.1 : BOOL;
    R101_2_I_RB_2차_작업완료 AT %MW84060.10 : BOOL;
    R101_2_I_RB_3차_간섭무 AT %MW84061.2 : BOOL;
    R101_2_I_RB_3차_작업완료 AT %MW84060.11 : BOOL;
    R101_2_I_RB_4차_간섭무 AT %MW84061.3 : BOOL;
    R101_2_I_RB_4차_작업완료 AT %MW84060.12 : BOOL;
    R101_2_I_RB_5차_간섭무 AT %MW84061.4 : BOOL;
    R101_2_I_RB_5차_작업완료 AT %MW84060.13 : BOOL;
    R101_2_I_RB_6차_간섭무 AT %MW84061.5 : BOOL;
    R101_2_I_RB_6차_작업완료 AT %MW84060.14 : BOOL;
    R101_2_I_RB_7차_간섭무 AT %MW84061.6 : BOOL;
    R101_2_I_RB_7차_작업완료 AT %MW84060.15 : BOOL;
    R101_2_I_RB_8차_간섭무 AT %MW84061.7 : BOOL;
    R101_2_I_RB_9차_간섭무 AT %MW84061.8 : BOOL;
    R101_2_I_RB_AB_NORMAL_선택 AT %MW84060.6 : BOOL;
    R101_2_I_RB_GUN1_FIXED_TIP AT %MW84067 : WORD;
    R101_2_I_RB_GUN1_MOVING_TIP AT %MW84066 : WORD;
    R101_2_I_RB_GUN2_FIXED_TIP AT %MW84069 : WORD;
    R101_2_I_RB_GUN2_MOVING_TIP AT %MW84068 : WORD;
    R101_2_I_RB_INPUT AT %MW84060 : ARRAY[0..3] OF WORD;
    R101_2_I_RB_LS_이상 AT %MW84062.11 : BOOL;
    R101_2_I_RB_MOTOR_MC_ON AT %MW84063.15 : BOOL;
    R101_2_I_RB_MUTUAL_INT1 AT %MW84063.0 : BOOL;
    R101_2_I_RB_MUTUAL_INT2 AT %MW84063.1 : BOOL;
    R101_2_I_RB_MUTUAL_INT3 AT %MW84063.2 : BOOL;
    R101_2_I_RB_MUTUAL_INT4 AT %MW84063.3 : BOOL;
    R101_2_I_RB_MUTUAL_INT5 AT %MW84063.4 : BOOL;
    R101_2_I_RB_MUTUAL_INT6 AT %MW84063.5 : BOOL;
    R101_2_I_RB_MUTUAL_INT7 AT %MW84063.6 : BOOL;
    R101_2_I_RB_MUTUAL_INT8 AT %MW84063.7 : BOOL;
    R101_2_I_RB_PLT_UNLOAD_완료 AT %MW84063.11 : BOOL;
    R101_2_I_RB_PLT_최종UNLOAD_완료 AT %MW84063.12 : BOOL;
    R101_2_I_RB_PROG_ECHO_1 AT %MW84062.0 : BOOL;
    R101_2_I_RB_PROG_ECHO_128 AT %MW84062.7 : BOOL;
    R101_2_I_RB_PROG_ECHO_16 AT %MW84062.4 : BOOL;
    R101_2_I_RB_PROG_ECHO_2 AT %MW84062.1 : BOOL;
    R101_2_I_RB_PROG_ECHO_32 AT %MW84062.5 : BOOL;
    R101_2_I_RB_PROG_ECHO_4 AT %MW84062.2 : BOOL;
    R101_2_I_RB_PROG_ECHO_64 AT %MW84062.6 : BOOL;
    R101_2_I_RB_PROG_ECHO_8 AT %MW84062.3 : BOOL;
    R101_2_I_RB_SP3_8 AT %MW84063.8 : BOOL;
    R101_2_I_RB_SP3_9 AT %MW84063.9 : BOOL;
    R101_2_I_RB_SPARE_WORD_4 AT %MW84064 : WORD;
    R101_2_I_RB_SP_1_12 AT %MW84061.12 : BOOL;
    R101_2_I_RB_SP_1_13 AT %MW84061.13 : BOOL;
    R101_2_I_RB_SP_1_14 AT %MW84061.14 : BOOL;
    R101_2_I_RB_SP_1_15 AT %MW84061.15 : BOOL;
    R101_2_I_RB_TC_이상 AT %MW84062.8 : BOOL;
    R101_2_I_RB_TIP_CHANGE AT %MW84063.13 : BOOL;
    R101_2_I_RB_TIP_DRESSING AT %MW84060.7 : BOOL;
    R101_2_I_RB__PLT_카운터리셋완료 AT %MW84063.10 : BOOL;
    R101_2_I_RB_공기압_이상 AT %MW84062.9 : BOOL;
    R101_2_I_RB_냉각수_이상 AT %MW84062.10 : BOOL;
    R101_2_I_RB_비상정지_NC AT %MW84060.8 : BOOL;
    R101_2_I_RB_비전이상 AT %MW84062.14 : BOOL;
    R101_2_I_RB_실러이상 AT %MW84062.13 : BOOL;
    R101_2_I_RB_용접카운터이상 AT %MW84062.15 : BOOL;
    R101_2_I_RB_용접타점수 AT %MW84065 : WORD;
    R101_2_I_RB_운전준비 AT %MW84060.3 : BOOL;
    R101_2_I_RB_원위치 AT %MW84060.0 : BOOL;
    R101_2_I_RB_이상리셋 AT %MW84060.2 : BOOL;
    R101_2_I_RB_자동 AT %MW84060.4 : BOOL;
    R101_2_I_RB_자동기동 AT %MW84060.5 : BOOL;
    R101_2_I_RB_최종_작업완료 AT %MW84060.1 : BOOL;
    R101_2_I_RB_통신이상 AT %MW84062.12 : BOOL;
    R101_2_M_AX_차종_용접타점수 AT %MW8120 : WORD; (* R101_2_M_AX_차종_용접타점수 *)
    R101_2_M_I_RB_1차_작업완료 AT %MW20061.2 : BOOL;
    R101_2_M_I_RB_2차_작업완료 AT %MW20061.3 : BOOL;
    R101_2_M_I_RB_3차_작업완료 AT %MW20061.4 : BOOL;
    R101_2_M_I_RB_4차_작업완료 AT %MW20061.5 : BOOL;
    R101_2_M_I_RB_5차_작업완료 AT %MW20061.6 : BOOL;
    R101_2_M_I_RB_6차_작업완료 AT %MW20061.7 : BOOL;
    R101_2_M_I_RB_7차_작업완료 AT %MW20061.8 : BOOL;
    R101_2_M_I_RB_PAUSE_보조 AT %MW20060.5 : BOOL;
    R101_2_M_I_RB_PLC_RUN_CHK_이상 AT %MW20060.7 : BOOL;
    R101_2_M_I_RB_간섭무_1 AT %MW20062.0 : BOOL;
    R101_2_M_I_RB_간섭무_10 AT %MW20062.9 : BOOL;
    R101_2_M_I_RB_간섭무_11 AT %MW20062.10 : BOOL;
    R101_2_M_I_RB_간섭무_12 AT %MW20062.11 : BOOL;
    R101_2_M_I_RB_간섭무_2 AT %MW20062.1 : BOOL;
    R101_2_M_I_RB_간섭무_3 AT %MW20062.2 : BOOL;
    R101_2_M_I_RB_간섭무_4 AT %MW20062.3 : BOOL;
    R101_2_M_I_RB_간섭무_5 AT %MW20062.4 : BOOL;
    R101_2_M_I_RB_간섭무_6 AT %MW20062.5 : BOOL;
    R101_2_M_I_RB_간섭무_7 AT %MW20062.6 : BOOL;
    R101_2_M_I_RB_간섭무_8 AT %MW20062.7 : BOOL;
    R101_2_M_I_RB_간섭무_9 AT %MW20062.8 : BOOL;
    R101_2_M_I_RB_비상정지 AT %MW20060.4 : BOOL;
    R101_2_M_I_RB_운전준비 AT %MW20060.0 : BOOL;
    R101_2_M_I_RB_원위치 AT %MW20060.3 : BOOL;
    R101_2_M_I_RB_이상 AT %MW20060.2 : BOOL;
    R101_2_M_I_RB_자동 AT %MW20060.1 : BOOL;
    R101_2_M_I_RB_최종작업완료 AT %MW20061.0 : BOOL;
    R101_2_M_I_RB_프로그램_이상 AT %MW20060.6 : BOOL;
    R101_2_M_O_RB_1_CYCLE_SET AT %MW21060.3 : BOOL;
    R101_2_M_O_RB_1_CYCLE_리셋 AT %MW21060.4 : BOOL;
    R101_2_M_O_RB_1차_작업완료_리셋 AT %MW21062.0 : BOOL;
    R101_2_M_O_RB_2차_작업완료_리셋 AT %MW21062.1 : BOOL;
    R101_2_M_O_RB_2차_진입OK AT %MW21061.8 : BOOL;
    R101_2_M_O_RB_3차_작업완료_리셋 AT %MW21062.2 : BOOL;
    R101_2_M_O_RB_3차_진입OK AT %MW21061.9 : BOOL;
    R101_2_M_O_RB_4차_작업완료_리셋 AT %MW21062.3 : BOOL;
    R101_2_M_O_RB_4차_진입OK AT %MW21061.10 : BOOL;
    R101_2_M_O_RB_5차_작업완료_리셋 AT %MW21062.4 : BOOL;
    R101_2_M_O_RB_5차_진입OK AT %MW21061.11 : BOOL;
    R101_2_M_O_RB_6차_작업완료_리셋 AT %MW21062.5 : BOOL;
    R101_2_M_O_RB_6차_진입OK AT %MW21061.12 : BOOL;
    R101_2_M_O_RB_7차_작업완료_리셋 AT %MW21062.6 : BOOL;
    R101_2_M_O_RB_7차_진입OK AT %MW21061.13 : BOOL;
    R101_2_M_O_RB_ATD_OK AT %MW21060.6 : BOOL;
    R101_2_M_O_RB_PLT_10_진입OK AT %MW21063.10 : BOOL;
    R101_2_M_O_RB_PLT_11_진입OK AT %MW21063.11 : BOOL;
    R101_2_M_O_RB_PLT_12_진입OK AT %MW21063.12 : BOOL;
    R101_2_M_O_RB_PLT_1_진입OK AT %MW21063.1 : BOOL;
    R101_2_M_O_RB_PLT_2_진입OK AT %MW21063.2 : BOOL;
    R101_2_M_O_RB_PLT_3_진입OK AT %MW21063.3 : BOOL;
    R101_2_M_O_RB_PLT_4_진입OK AT %MW21063.4 : BOOL;
    R101_2_M_O_RB_PLT_5_진입OK AT %MW21063.5 : BOOL;
    R101_2_M_O_RB_PLT_6_진입OK AT %MW21063.6 : BOOL;
    R101_2_M_O_RB_PLT_7_진입OK AT %MW21063.7 : BOOL;
    R101_2_M_O_RB_PLT_8_진입OK AT %MW21063.8 : BOOL;
    R101_2_M_O_RB_PLT_9_진입OK AT %MW21063.9 : BOOL;
    R101_2_M_O_RB_PLT_카운터리셋_보조 AT %MW21060.10 : BOOL;
    R101_2_M_O_RB_RESTART_OK AT %MW21060.2 : BOOL;
    R101_2_M_O_RB_START_OK AT %MW21060.0 : BOOL;
    R101_2_M_O_RB_TEST_MODE_5000회 AT %MW21060.12 : BOOL;
    R101_2_M_O_RB_TIP_교체_시작 AT %MW21060.7 : BOOL;
    R101_2_M_O_RB_TIP_교체_완료 AT %MW21060.8 : BOOL;
    R101_2_M_O_RB_VIP_MODE AT %MW21060.11 : BOOL;
    R101_2_M_O_RB_냉각수_차단_요청 AT %MW21060.9 : BOOL;
    R101_2_M_O_RB_진입OK_AX차종 AT %MW21061.0 : BOOL;
    R101_2_M_O_RB_진입OK_B차종 AT %MW21061.1 : BOOL;
    R101_2_M_O_RB_진입OK_C차종 AT %MW21061.2 : BOOL;
    R101_2_M_O_RB_진입OK_D차종 AT %MW21061.3 : BOOL;
    R101_2_M_O_RB_진입OK_E차종 AT %MW21061.4 : BOOL;
    R101_2_M_O_RB_진입OK_F차종 AT %MW21061.5 : BOOL;
    R101_2_M_O_RB_진입OK_G차종 AT %MW21061.6 : BOOL;
    R101_2_M_O_RB_진입OK_H차종 AT %MW21061.7 : BOOL;
    R101_2_M_O_RB_최종_작업완료_리셋 AT %MW21060.5 : BOOL;
    R101_2_M_O_RB_프로그램_OK AT %MW21060.1 : BOOL;
    R101_2_M_RB_PROG_NO AT %MW20064 : WORD;
    R101_2_M_RB_통신이상 AT %MW1024.12 : BOOL;
    R101_2_M_용접완료 AT %MW1011.2 : BOOL;
    R101_2_M_용접타점수_OK AT %MW1011.6 : BOOL;
    R101_2_M_용접타점수_이상 AT %MW1011.11 : BOOL;
    R101_2_O_RB_0_5S_통신_CHK AT %MW94063.14 : BOOL;
    R101_2_O_RB_2차_진입OK AT %MW94061.8 : BOOL;
    R101_2_O_RB_3차_진입OK AT %MW94061.9 : BOOL;
    R101_2_O_RB_4차_진입OK AT %MW94061.10 : BOOL;
    R101_2_O_RB_5차_진입OK AT %MW94061.11 : BOOL;
    R101_2_O_RB_6차_진입OK AT %MW94061.12 : BOOL;
    R101_2_O_RB_7차_진입OK AT %MW94061.13 : BOOL;
    R101_2_O_RB_AX_1차_진입OK AT %MW94061.0 : BOOL;
    R101_2_O_RB_B_1차_진입OK AT %MW94061.1 : BOOL;
    R101_2_O_RB_C_1차_진입OK AT %MW94061.2 : BOOL;
    R101_2_O_RB_D_1차_진입OK AT %MW94061.3 : BOOL;
    R101_2_O_RB_EACH_작업완료_리셋 AT %MW94060.14 : BOOL;
    R101_2_O_RB_EXT_READY AT %MW94060.11 : BOOL;
    R101_2_O_RB_E_1차_진입OK AT %MW94061.4 : BOOL;
    R101_2_O_RB_F_1차_진입OK AT %MW94061.5 : BOOL;
    R101_2_O_RB_GATE_OPEN_NC AT %MW94063.11 : BOOL;
    R101_2_O_RB_G_1차_진입OK AT %MW94061.6 : BOOL;
    R101_2_O_RB_H_1차_진입OK AT %MW94061.7 : BOOL;
    R101_2_O_RB_MUTUAL_INT1 AT %MW94063.0 : BOOL;
    R101_2_O_RB_MUTUAL_INT2 AT %MW94063.1 : BOOL;
    R101_2_O_RB_MUTUAL_INT3 AT %MW94063.2 : BOOL;
    R101_2_O_RB_MUTUAL_INT4 AT %MW94063.3 : BOOL;
    R101_2_O_RB_MUTUAL_INT5 AT %MW94063.4 : BOOL;
    R101_2_O_RB_MUTUAL_INT6 AT %MW94063.5 : BOOL;
    R101_2_O_RB_MUTUAL_INT7 AT %MW94063.6 : BOOL;
    R101_2_O_RB_MUTUAL_INT8 AT %MW94063.7 : BOOL;
    R101_2_O_RB_OUTPUT AT %MW94060 : ARRAY[0..3] OF WORD;
    R101_2_O_RB_PAUSE_NC AT %MW94060.13 : BOOL;
    R101_2_O_RB_PLT10_진입OK AT %MW94062.9 : BOOL;
    R101_2_O_RB_PLT11_진입OK AT %MW94062.10 : BOOL;
    R101_2_O_RB_PLT12_진입OK AT %MW94062.11 : BOOL;
    R101_2_O_RB_PLT1_진입OK AT %MW94062.0 : BOOL;
    R101_2_O_RB_PLT2_진입OK AT %MW94062.1 : BOOL;
    R101_2_O_RB_PLT3_진입OK AT %MW94062.2 : BOOL;
    R101_2_O_RB_PLT4_진입OK AT %MW94062.3 : BOOL;
    R101_2_O_RB_PLT5_진입OK AT %MW94062.4 : BOOL;
    R101_2_O_RB_PLT6_진입OK AT %MW94062.5 : BOOL;
    R101_2_O_RB_PLT7_진입OK AT %MW94062.6 : BOOL;
    R101_2_O_RB_PLT8_진입OK AT %MW94062.7 : BOOL;
    R101_2_O_RB_PLT9_진입OK AT %MW94062.8 : BOOL;
    R101_2_O_RB_PLT_COUNT_리셋_COND AT %MW94063.10 : BOOL;
    R101_2_O_RB_PROG_선택1 AT %MW94060.0 : BOOL;
    R101_2_O_RB_PROG_선택128 AT %MW94060.7 : BOOL;
    R101_2_O_RB_PROG_선택16 AT %MW94060.4 : BOOL;
    R101_2_O_RB_PROG_선택2 AT %MW94060.1 : BOOL;
    R101_2_O_RB_PROG_선택32 AT %MW94060.5 : BOOL;
    R101_2_O_RB_PROG_선택4 AT %MW94060.2 : BOOL;
    R101_2_O_RB_PROG_선택64 AT %MW94060.6 : BOOL;
    R101_2_O_RB_PROG_선택8 AT %MW94060.3 : BOOL;
    R101_2_O_RB_SP_1_14 AT %MW94061.14 : BOOL;
    R101_2_O_RB_SP_1_15 AT %MW94061.15 : BOOL;
    R101_2_O_RB_SP_2_12 AT %MW94062.12 : BOOL;
    R101_2_O_RB_SP_2_13 AT %MW94062.13 : BOOL;
    R101_2_O_RB_SP_2_14 AT %MW94062.14 : BOOL;
    R101_2_O_RB_SP_5000TH_ON AT %MW94062.15 : BOOL;
    R101_2_O_RB_TIP_CHANGE_END AT %MW94063.9 : BOOL;
    R101_2_O_RB_TIP_CHANGE_START AT %MW94063.8 : BOOL;
    R101_2_O_RB_TIP_DRESS_SATRT AT %MW94060.12 : BOOL;
    R101_2_O_RB_VIP_MODE AT %MW94063.15 : BOOL;
    R101_2_O_RB_기동 AT %MW94060.9 : BOOL;
    R101_2_O_RB_냉각수차단 AT %MW94060.15 : BOOL;
    R101_2_O_RB_부저정지 AT %MW94063.13 : BOOL;
    R101_2_O_RB_비상정지_NC AT %MW94063.12 : BOOL;
    R101_2_O_RB_이상_리셋 AT %MW94060.10 : BOOL;
    R101_2_O_RB_작업완료_리셋 AT %MW94060.8 : BOOL;
    R101_3_I_RB_0_5_COMM_CHK AT %MW84053.14 : BOOL;
    R101_3_I_RB_10차_간섭무 AT %MW84051.9 : BOOL;
    R101_3_I_RB_11차_간섭무 AT %MW84051.10 : BOOL;
    R101_3_I_RB_12차_간섭무 AT %MW84051.11 : BOOL;
    R101_3_I_RB_1차_간섭무 AT %MW84051.0 : BOOL;
    R101_3_I_RB_1차_작업완료 AT %MW84050.9 : BOOL;
    R101_3_I_RB_2차_간섭무 AT %MW84051.1 : BOOL;
    R101_3_I_RB_2차_작업완료 AT %MW84050.10 : BOOL;
    R101_3_I_RB_3차_간섭무 AT %MW84051.2 : BOOL;
    R101_3_I_RB_3차_작업완료 AT %MW84050.11 : BOOL;
    R101_3_I_RB_4차_간섭무 AT %MW84051.3 : BOOL;
    R101_3_I_RB_4차_작업완료 AT %MW84050.12 : BOOL;
    R101_3_I_RB_5차_간섭무 AT %MW84051.4 : BOOL;
    R101_3_I_RB_5차_작업완료 AT %MW84050.13 : BOOL;
    R101_3_I_RB_6차_간섭무 AT %MW84051.5 : BOOL;
    R101_3_I_RB_6차_작업완료 AT %MW84050.14 : BOOL;
    R101_3_I_RB_7차_간섭무 AT %MW84051.6 : BOOL;
    R101_3_I_RB_7차_작업완료 AT %MW84050.15 : BOOL;
    R101_3_I_RB_8차_간섭무 AT %MW84051.7 : BOOL;
    R101_3_I_RB_9차_간섭무 AT %MW84051.8 : BOOL;
    R101_3_I_RB_AB_NORMAL_선택 AT %MW84050.6 : BOOL;
    R101_3_I_RB_GUN1_FIXED_TIP AT %MW84057 : WORD;
    R101_3_I_RB_GUN1_MOVING_TIP AT %MW84056 : WORD;
    R101_3_I_RB_GUN2_FIXED_TIP AT %MW84059 : WORD;
    R101_3_I_RB_GUN2_MOVING_TIP AT %MW84058 : WORD;
    R101_3_I_RB_INPUT AT %MW84050 : ARRAY[0..3] OF WORD;
    R101_3_I_RB_LS_이상 AT %MW84052.11 : BOOL;
    R101_3_I_RB_MOTOR_MC_ON AT %MW84053.15 : BOOL;
    R101_3_I_RB_MUTUAL_INT1 AT %MW84053.0 : BOOL;
    R101_3_I_RB_MUTUAL_INT2 AT %MW84053.1 : BOOL;
    R101_3_I_RB_MUTUAL_INT3 AT %MW84053.2 : BOOL;
    R101_3_I_RB_MUTUAL_INT4 AT %MW84053.3 : BOOL;
    R101_3_I_RB_MUTUAL_INT5 AT %MW84053.4 : BOOL;
    R101_3_I_RB_MUTUAL_INT6 AT %MW84053.5 : BOOL;
    R101_3_I_RB_MUTUAL_INT7 AT %MW84053.6 : BOOL;
    R101_3_I_RB_MUTUAL_INT8 AT %MW84053.7 : BOOL;
    R101_3_I_RB_PLT_UNLOAD_완료 AT %MW84053.11 : BOOL;
    R101_3_I_RB_PLT_최종UNLOAD_완료 AT %MW84053.12 : BOOL;
    R101_3_I_RB_PROG_ECHO_1 AT %MW84052.0 : BOOL;
    R101_3_I_RB_PROG_ECHO_128 AT %MW84052.7 : BOOL;
    R101_3_I_RB_PROG_ECHO_16 AT %MW84052.4 : BOOL;
    R101_3_I_RB_PROG_ECHO_2 AT %MW84052.1 : BOOL;
    R101_3_I_RB_PROG_ECHO_32 AT %MW84052.5 : BOOL;
    R101_3_I_RB_PROG_ECHO_4 AT %MW84052.2 : BOOL;
    R101_3_I_RB_PROG_ECHO_64 AT %MW84052.6 : BOOL;
    R101_3_I_RB_PROG_ECHO_8 AT %MW84052.3 : BOOL;
    R101_3_I_RB_SP3_8 AT %MW84053.8 : BOOL;
    R101_3_I_RB_SP3_9 AT %MW84053.9 : BOOL;
    R101_3_I_RB_SPARE_WORD_4 AT %MW84054 : WORD;
    R101_3_I_RB_SP_1_12 AT %MW84051.12 : BOOL;
    R101_3_I_RB_SP_1_13 AT %MW84051.13 : BOOL;
    R101_3_I_RB_SP_1_14 AT %MW84051.14 : BOOL;
    R101_3_I_RB_SP_1_15 AT %MW84051.15 : BOOL;
    R101_3_I_RB_TC_이상 AT %MW84052.8 : BOOL;
    R101_3_I_RB_TIP_CHANGE AT %MW84053.13 : BOOL;
    R101_3_I_RB_TIP_DRESSING AT %MW84050.7 : BOOL;
    R101_3_I_RB__PLT_카운터리셋완료 AT %MW84053.10 : BOOL;
    R101_3_I_RB_공기압_이상 AT %MW84052.9 : BOOL;
    R101_3_I_RB_냉각수_이상 AT %MW84052.10 : BOOL;
    R101_3_I_RB_비상정지_NC AT %MW84050.8 : BOOL;
    R101_3_I_RB_비전이상 AT %MW84052.14 : BOOL;
    R101_3_I_RB_실러이상 AT %MW84052.13 : BOOL;
    R101_3_I_RB_용접카운터이상 AT %MW84052.15 : BOOL;
    R101_3_I_RB_용접타점수 AT %MW84055 : WORD;
    R101_3_I_RB_운전준비 AT %MW84050.3 : BOOL;
    R101_3_I_RB_원위치 AT %MW84050.0 : BOOL;
    R101_3_I_RB_이상리셋 AT %MW84050.2 : BOOL;
    R101_3_I_RB_자동 AT %MW84050.4 : BOOL;
    R101_3_I_RB_자동기동 AT %MW84050.5 : BOOL;
    R101_3_I_RB_최종_작업완료 AT %MW84050.1 : BOOL;
    R101_3_I_RB_통신이상 AT %MW84052.12 : BOOL;
    R101_3_M_I_RB_1차_작업완료 AT %MW20051.2 : BOOL;
    R101_3_M_I_RB_2차_작업완료 AT %MW20051.3 : BOOL;
    R101_3_M_I_RB_3차_작업완료 AT %MW20051.4 : BOOL;
    R101_3_M_I_RB_4차_작업완료 AT %MW20051.5 : BOOL;
    R101_3_M_I_RB_5차_작업완료 AT %MW20051.6 : BOOL;
    R101_3_M_I_RB_6차_작업완료 AT %MW20051.7 : BOOL;
    R101_3_M_I_RB_7차_작업완료 AT %MW20051.8 : BOOL;
    R101_3_M_I_RB_PAUSE_보조 AT %MW20050.5 : BOOL;
    R101_3_M_I_RB_PLC_RUN_CHK_이상 AT %MW20050.7 : BOOL;
    R101_3_M_I_RB_간섭무_1 AT %MW20052.0 : BOOL;
    R101_3_M_I_RB_간섭무_10 AT %MW20052.9 : BOOL;
    R101_3_M_I_RB_간섭무_11 AT %MW20052.10 : BOOL;
    R101_3_M_I_RB_간섭무_12 AT %MW20052.11 : BOOL;
    R101_3_M_I_RB_간섭무_2 AT %MW20052.1 : BOOL;
    R101_3_M_I_RB_간섭무_3 AT %MW20052.2 : BOOL;
    R101_3_M_I_RB_간섭무_4 AT %MW20052.3 : BOOL;
    R101_3_M_I_RB_간섭무_5 AT %MW20052.4 : BOOL;
    R101_3_M_I_RB_간섭무_6 AT %MW20052.5 : BOOL;
    R101_3_M_I_RB_간섭무_7 AT %MW20052.6 : BOOL;
    R101_3_M_I_RB_간섭무_8 AT %MW20052.7 : BOOL;
    R101_3_M_I_RB_간섭무_9 AT %MW20052.8 : BOOL;
    R101_3_M_I_RB_비상정지 AT %MW20050.4 : BOOL;
    R101_3_M_I_RB_운전준비 AT %MW20050.0 : BOOL;
    R101_3_M_I_RB_원위치 AT %MW20050.3 : BOOL;
    R101_3_M_I_RB_이상 AT %MW20050.2 : BOOL;
    R101_3_M_I_RB_자동 AT %MW20050.1 : BOOL;
    R101_3_M_I_RB_최종작업완료 AT %MW20051.0 : BOOL;
    R101_3_M_I_RB_프로그램_이상 AT %MW20050.6 : BOOL;
    R101_3_M_O_RB_1_CYCLE_SET AT %MW21050.3 : BOOL;
    R101_3_M_O_RB_1_CYCLE_리셋 AT %MW21050.4 : BOOL;
    R101_3_M_O_RB_1차_작업완료_리셋 AT %MW21052.0 : BOOL;
    R101_3_M_O_RB_2차_작업완료_리셋 AT %MW21052.1 : BOOL;
    R101_3_M_O_RB_2차_진입OK AT %MW21051.8 : BOOL;
    R101_3_M_O_RB_3차_작업완료_리셋 AT %MW21052.2 : BOOL;
    R101_3_M_O_RB_3차_진입OK AT %MW21051.9 : BOOL;
    R101_3_M_O_RB_4차_작업완료_리셋 AT %MW21052.3 : BOOL;
    R101_3_M_O_RB_4차_진입OK AT %MW21051.10 : BOOL;
    R101_3_M_O_RB_5차_작업완료_리셋 AT %MW21052.4 : BOOL;
    R101_3_M_O_RB_5차_진입OK AT %MW21051.11 : BOOL;
    R101_3_M_O_RB_6차_작업완료_리셋 AT %MW21052.5 : BOOL;
    R101_3_M_O_RB_6차_진입OK AT %MW21051.12 : BOOL;
    R101_3_M_O_RB_7차_작업완료_리셋 AT %MW21052.6 : BOOL;
    R101_3_M_O_RB_7차_진입OK AT %MW21051.13 : BOOL;
    R101_3_M_O_RB_ATD_OK AT %MW21050.6 : BOOL;
    R101_3_M_O_RB_PLT_10_진입OK AT %MW21053.10 : BOOL;
    R101_3_M_O_RB_PLT_11_진입OK AT %MW21053.11 : BOOL;
    R101_3_M_O_RB_PLT_12_진입OK AT %MW21053.12 : BOOL;
    R101_3_M_O_RB_PLT_1_진입OK AT %MW21053.1 : BOOL;
    R101_3_M_O_RB_PLT_2_진입OK AT %MW21053.2 : BOOL;
    R101_3_M_O_RB_PLT_3_진입OK AT %MW21053.3 : BOOL;
    R101_3_M_O_RB_PLT_4_진입OK AT %MW21053.4 : BOOL;
    R101_3_M_O_RB_PLT_5_진입OK AT %MW21053.5 : BOOL;
    R101_3_M_O_RB_PLT_6_진입OK AT %MW21053.6 : BOOL;
    R101_3_M_O_RB_PLT_7_진입OK AT %MW21053.7 : BOOL;
    R101_3_M_O_RB_PLT_8_진입OK AT %MW21053.8 : BOOL;
    R101_3_M_O_RB_PLT_9_진입OK AT %MW21053.9 : BOOL;
    R101_3_M_O_RB_PLT_카운터리셋_보조 AT %MW21050.10 : BOOL;
    R101_3_M_O_RB_RESTART_OK AT %MW21050.2 : BOOL;
    R101_3_M_O_RB_START_OK AT %MW21050.0 : BOOL;
    R101_3_M_O_RB_TEST_MODE_5000회 AT %MW21050.12 : BOOL;
    R101_3_M_O_RB_TIP_교체_시작 AT %MW21050.7 : BOOL;
    R101_3_M_O_RB_TIP_교체_완료 AT %MW21050.8 : BOOL;
    R101_3_M_O_RB_VIP_MODE AT %MW21050.11 : BOOL;
    R101_3_M_O_RB_냉각수_차단_요청 AT %MW21050.9 : BOOL;
    R101_3_M_O_RB_진입OK_AX차종 AT %MW21051.0 : BOOL;
    R101_3_M_O_RB_진입OK_B차종 AT %MW21051.1 : BOOL;
    R101_3_M_O_RB_진입OK_C차종 AT %MW21051.2 : BOOL;
    R101_3_M_O_RB_진입OK_D차종 AT %MW21051.3 : BOOL;
    R101_3_M_O_RB_진입OK_E차종 AT %MW21051.4 : BOOL;
    R101_3_M_O_RB_진입OK_F차종 AT %MW21051.5 : BOOL;
    R101_3_M_O_RB_진입OK_G차종 AT %MW21051.6 : BOOL;
    R101_3_M_O_RB_진입OK_H차종 AT %MW21051.7 : BOOL;
    R101_3_M_O_RB_최종_작업완료_리셋 AT %MW21050.5 : BOOL;
    R101_3_M_O_RB_프로그램_OK AT %MW21050.1 : BOOL;
    R101_3_M_RB_PROG_NO AT %MW20054 : WORD;
    R101_3_M_RB_통신이상 AT %MW1024.13 : BOOL;
    R101_3_O_RB_0_5S_통신_CHK AT %MW94053.14 : BOOL;
    R101_3_O_RB_2차_진입OK AT %MW94051.8 : BOOL;
    R101_3_O_RB_3차_진입OK AT %MW94051.9 : BOOL;
    R101_3_O_RB_4차_진입OK AT %MW94051.10 : BOOL;
    R101_3_O_RB_5차_진입OK AT %MW94051.11 : BOOL;
    R101_3_O_RB_6차_진입OK AT %MW94051.12 : BOOL;
    R101_3_O_RB_7차_진입OK AT %MW94051.13 : BOOL;
    R101_3_O_RB_AX_1차_진입OK AT %MW94051.0 : BOOL;
    R101_3_O_RB_B_1차_진입OK AT %MW94051.1 : BOOL;
    R101_3_O_RB_C_1차_진입OK AT %MW94051.2 : BOOL;
    R101_3_O_RB_D_1차_진입OK AT %MW94051.3 : BOOL;
    R101_3_O_RB_EACH_작업완료_리셋 AT %MW94050.14 : BOOL;
    R101_3_O_RB_EXT_READY AT %MW94050.11 : BOOL;
    R101_3_O_RB_E_1차_진입OK AT %MW94051.4 : BOOL;
    R101_3_O_RB_F_1차_진입OK AT %MW94051.5 : BOOL;
    R101_3_O_RB_GATE_OPEN_NC AT %MW94053.11 : BOOL;
    R101_3_O_RB_G_1차_진입OK AT %MW94051.6 : BOOL;
    R101_3_O_RB_H_1차_진입OK AT %MW94051.7 : BOOL;
    R101_3_O_RB_MUTUAL_INT1 AT %MW94053.0 : BOOL;
    R101_3_O_RB_MUTUAL_INT2 AT %MW94053.1 : BOOL;
    R101_3_O_RB_MUTUAL_INT3 AT %MW94053.2 : BOOL;
    R101_3_O_RB_MUTUAL_INT4 AT %MW94053.3 : BOOL;
    R101_3_O_RB_MUTUAL_INT5 AT %MW94053.4 : BOOL;
    R101_3_O_RB_MUTUAL_INT6 AT %MW94053.5 : BOOL;
    R101_3_O_RB_MUTUAL_INT7 AT %MW94053.6 : BOOL;
    R101_3_O_RB_MUTUAL_INT8 AT %MW94053.7 : BOOL;
    R101_3_O_RB_OUTPUT AT %MW94050 : ARRAY[0..3] OF WORD;
    R101_3_O_RB_PAUSE_NC AT %MW94050.13 : BOOL;
    R101_3_O_RB_PLT10_진입OK AT %MW94052.9 : BOOL;
    R101_3_O_RB_PLT11_진입OK AT %MW94052.10 : BOOL;
    R101_3_O_RB_PLT12_진입OK AT %MW94052.11 : BOOL;
    R101_3_O_RB_PLT1_진입OK AT %MW94052.0 : BOOL;
    R101_3_O_RB_PLT2_진입OK AT %MW94052.1 : BOOL;
    R101_3_O_RB_PLT3_진입OK AT %MW94052.2 : BOOL;
    R101_3_O_RB_PLT4_진입OK AT %MW94052.3 : BOOL;
    R101_3_O_RB_PLT5_진입OK AT %MW94052.4 : BOOL;
    R101_3_O_RB_PLT6_진입OK AT %MW94052.5 : BOOL;
    R101_3_O_RB_PLT7_진입OK AT %MW94052.6 : BOOL;
    R101_3_O_RB_PLT8_진입OK AT %MW94052.7 : BOOL;
    R101_3_O_RB_PLT9_진입OK AT %MW94052.8 : BOOL;
    R101_3_O_RB_PLT_COUNT_리셋_COND AT %MW94053.10 : BOOL;
    R101_3_O_RB_PROG_선택1 AT %MW94050.0 : BOOL;
    R101_3_O_RB_PROG_선택128 AT %MW94050.7 : BOOL;
    R101_3_O_RB_PROG_선택16 AT %MW94050.4 : BOOL;
    R101_3_O_RB_PROG_선택2 AT %MW94050.1 : BOOL;
    R101_3_O_RB_PROG_선택32 AT %MW94050.5 : BOOL;
    R101_3_O_RB_PROG_선택4 AT %MW94050.2 : BOOL;
    R101_3_O_RB_PROG_선택64 AT %MW94050.6 : BOOL;
    R101_3_O_RB_PROG_선택8 AT %MW94050.3 : BOOL;
    R101_3_O_RB_SP_1_14 AT %MW94051.14 : BOOL;
    R101_3_O_RB_SP_1_15 AT %MW94051.15 : BOOL;
    R101_3_O_RB_SP_2_12 AT %MW94052.12 : BOOL;
    R101_3_O_RB_SP_2_13 AT %MW94052.13 : BOOL;
    R101_3_O_RB_SP_2_14 AT %MW94052.14 : BOOL;
    R101_3_O_RB_SP_5000TH_ON AT %MW94052.15 : BOOL;
    R101_3_O_RB_TIP_CHANGE_END AT %MW94053.9 : BOOL;
    R101_3_O_RB_TIP_CHANGE_START AT %MW94053.8 : BOOL;
    R101_3_O_RB_TIP_DRESS_SATRT AT %MW94050.12 : BOOL;
    R101_3_O_RB_VIP_MODE AT %MW94053.15 : BOOL;
    R101_3_O_RB_기동 AT %MW94050.9 : BOOL;
    R101_3_O_RB_냉각수차단 AT %MW94050.15 : BOOL;
    R101_3_O_RB_부저정지 AT %MW94053.13 : BOOL;
    R101_3_O_RB_비상정지_NC AT %MW94053.12 : BOOL;
    R101_3_O_RB_이상_리셋 AT %MW94050.10 : BOOL;
    R101_3_O_RB_작업완료_리셋 AT %MW94050.8 : BOOL;
    R101_3축_리어_I_RB_0_5_COMM_CHK AT %MW84033.14 : BOOL;
    R101_3축_리어_I_RB_10차_간섭무 AT %MW84031.9 : BOOL;
    R101_3축_리어_I_RB_11차_간섭무 AT %MW84031.10 : BOOL;
    R101_3축_리어_I_RB_12차_간섭무 AT %MW84031.11 : BOOL;
    R101_3축_리어_I_RB_1차_간섭무 AT %MW84031.0 : BOOL;
    R101_3축_리어_I_RB_1차_작업완료 AT %MW84030.9 : BOOL;
    R101_3축_리어_I_RB_2차_간섭무 AT %MW84031.1 : BOOL;
    R101_3축_리어_I_RB_2차_작업완료 AT %MW84030.10 : BOOL;
    R101_3축_리어_I_RB_3차_간섭무 AT %MW84031.2 : BOOL;
    R101_3축_리어_I_RB_3차_작업완료 AT %MW84030.11 : BOOL;
    R101_3축_리어_I_RB_4차_간섭무 AT %MW84031.3 : BOOL;
    R101_3축_리어_I_RB_4차_작업완료 AT %MW84030.12 : BOOL;
    R101_3축_리어_I_RB_5차_간섭무 AT %MW84031.4 : BOOL;
    R101_3축_리어_I_RB_5차_작업완료 AT %MW84030.13 : BOOL;
    R101_3축_리어_I_RB_6차_간섭무 AT %MW84031.5 : BOOL;
    R101_3축_리어_I_RB_6차_작업완료 AT %MW84030.14 : BOOL;
    R101_3축_리어_I_RB_7차_간섭무 AT %MW84031.6 : BOOL;
    R101_3축_리어_I_RB_7차_작업완료 AT %MW84030.15 : BOOL;
    R101_3축_리어_I_RB_8차_간섭무 AT %MW84031.7 : BOOL;
    R101_3축_리어_I_RB_9차_간섭무 AT %MW84031.8 : BOOL;
    R101_3축_리어_I_RB_AB_NORMAL_선택 AT %MW84030.6 : BOOL;
    R101_3축_리어_I_RB_GUN1_FIXED_TIP AT %MW84037 : WORD;
    R101_3축_리어_I_RB_GUN1_MOVING_TIP AT %MW84036 : WORD;
    R101_3축_리어_I_RB_GUN2_FIXED_TIP AT %MW84039 : WORD;
    R101_3축_리어_I_RB_GUN2_MOVING_TIP AT %MW84038 : WORD;
    R101_3축_리어_I_RB_INPUT AT %MW84030 : ARRAY[0..3] OF WORD;
    R101_3축_리어_I_RB_LS_이상 AT %MW84032.11 : BOOL;
    R101_3축_리어_I_RB_MOTOR_MC_ON AT %MW84033.15 : BOOL;
    R101_3축_리어_I_RB_MUTUAL_INT1 AT %MW84033.0 : BOOL;
    R101_3축_리어_I_RB_MUTUAL_INT2 AT %MW84033.1 : BOOL;
    R101_3축_리어_I_RB_MUTUAL_INT3 AT %MW84033.2 : BOOL;
    R101_3축_리어_I_RB_MUTUAL_INT4 AT %MW84033.3 : BOOL;
    R101_3축_리어_I_RB_MUTUAL_INT5 AT %MW84033.4 : BOOL;
    R101_3축_리어_I_RB_MUTUAL_INT6 AT %MW84033.5 : BOOL;
    R101_3축_리어_I_RB_MUTUAL_INT7 AT %MW84033.6 : BOOL;
    R101_3축_리어_I_RB_MUTUAL_INT8 AT %MW84033.7 : BOOL;
    R101_3축_리어_I_RB_PLT_UNLOAD_완료 AT %MW84033.11 : BOOL;
    R101_3축_리어_I_RB_PLT_최종UNLOAD_완료 AT %MW84033.12 : BOOL;
    R101_3축_리어_I_RB_PROG_ECHO_1 AT %MW84032.0 : BOOL;
    R101_3축_리어_I_RB_PROG_ECHO_128 AT %MW84032.7 : BOOL;
    R101_3축_리어_I_RB_PROG_ECHO_16 AT %MW84032.4 : BOOL;
    R101_3축_리어_I_RB_PROG_ECHO_2 AT %MW84032.1 : BOOL;
    R101_3축_리어_I_RB_PROG_ECHO_32 AT %MW84032.5 : BOOL;
    R101_3축_리어_I_RB_PROG_ECHO_4 AT %MW84032.2 : BOOL;
    R101_3축_리어_I_RB_PROG_ECHO_64 AT %MW84032.6 : BOOL;
    R101_3축_리어_I_RB_PROG_ECHO_8 AT %MW84032.3 : BOOL;
    R101_3축_리어_I_RB_SP3_8 AT %MW84033.8 : BOOL;
    R101_3축_리어_I_RB_SP3_9 AT %MW84033.9 : BOOL;
    R101_3축_리어_I_RB_SPARE_WORD_4 AT %MW84034 : WORD;
    R101_3축_리어_I_RB_SP_1_12 AT %MW84031.12 : BOOL;
    R101_3축_리어_I_RB_SP_1_13 AT %MW84031.13 : BOOL;
    R101_3축_리어_I_RB_SP_1_14 AT %MW84031.14 : BOOL;
    R101_3축_리어_I_RB_SP_1_15 AT %MW84031.15 : BOOL;
    R101_3축_리어_I_RB_TC_이상 AT %MW84032.8 : BOOL;
    R101_3축_리어_I_RB_TIP_CHANGE AT %MW84033.13 : BOOL;
    R101_3축_리어_I_RB_TIP_DRESSING AT %MW84030.7 : BOOL;
    R101_3축_리어_I_RB__PLT_카운터리셋완료 AT %MW84033.10 : BOOL;
    R101_3축_리어_I_RB_공기압_이상 AT %MW84032.9 : BOOL;
    R101_3축_리어_I_RB_냉각수_이상 AT %MW84032.10 : BOOL;
    R101_3축_리어_I_RB_비상정지_NC AT %MW84030.8 : BOOL;
    R101_3축_리어_I_RB_비전이상 AT %MW84032.14 : BOOL;
    R101_3축_리어_I_RB_실러이상 AT %MW84032.13 : BOOL;
    R101_3축_리어_I_RB_용접카운터이상 AT %MW84032.15 : BOOL;
    R101_3축_리어_I_RB_용접타점수 AT %MW84035 : WORD;
    R101_3축_리어_I_RB_운전준비 AT %MW84030.3 : BOOL;
    R101_3축_리어_I_RB_원위치 AT %MW84030.0 : BOOL;
    R101_3축_리어_I_RB_이상리셋 AT %MW84030.2 : BOOL;
    R101_3축_리어_I_RB_자동 AT %MW84030.4 : BOOL;
    R101_3축_리어_I_RB_자동기동 AT %MW84030.5 : BOOL;
    R101_3축_리어_I_RB_최종_작업완료 AT %MW84030.1 : BOOL;
    R101_3축_리어_I_RB_통신이상 AT %MW84032.12 : BOOL;
    R101_3축_리어_M_I_RB_1차_작업완료 AT %MW20031.2 : BOOL;
    R101_3축_리어_M_I_RB_2차_작업완료 AT %MW20031.3 : BOOL;
    R101_3축_리어_M_I_RB_3차_작업완료 AT %MW20031.4 : BOOL;
    R101_3축_리어_M_I_RB_4차_작업완료 AT %MW20031.5 : BOOL;
    R101_3축_리어_M_I_RB_5차_작업완료 AT %MW20031.6 : BOOL;
    R101_3축_리어_M_I_RB_6차_작업완료 AT %MW20031.7 : BOOL;
    R101_3축_리어_M_I_RB_7차_작업완료 AT %MW20031.8 : BOOL;
    R101_3축_리어_M_I_RB_PAUSE_보조 AT %MW20030.5 : BOOL;
    R101_3축_리어_M_I_RB_PLC_RUN_CHK_이상 AT %MW20030.7 : BOOL;
    R101_3축_리어_M_I_RB_간섭무_1 AT %MW20032.0 : BOOL;
    R101_3축_리어_M_I_RB_간섭무_10 AT %MW20032.9 : BOOL;
    R101_3축_리어_M_I_RB_간섭무_11 AT %MW20032.10 : BOOL;
    R101_3축_리어_M_I_RB_간섭무_12 AT %MW20032.11 : BOOL;
    R101_3축_리어_M_I_RB_간섭무_2 AT %MW20032.1 : BOOL;
    R101_3축_리어_M_I_RB_간섭무_3 AT %MW20032.2 : BOOL;
    R101_3축_리어_M_I_RB_간섭무_4 AT %MW20032.3 : BOOL;
    R101_3축_리어_M_I_RB_간섭무_5 AT %MW20032.4 : BOOL;
    R101_3축_리어_M_I_RB_간섭무_6 AT %MW20032.5 : BOOL;
    R101_3축_리어_M_I_RB_간섭무_7 AT %MW20032.6 : BOOL;
    R101_3축_리어_M_I_RB_간섭무_8 AT %MW20032.7 : BOOL;
    R101_3축_리어_M_I_RB_간섭무_9 AT %MW20032.8 : BOOL;
    R101_3축_리어_M_I_RB_비상정지 AT %MW20030.4 : BOOL;
    R101_3축_리어_M_I_RB_운전준비 AT %MW20030.0 : BOOL;
    R101_3축_리어_M_I_RB_원위치 AT %MW20030.3 : BOOL;
    R101_3축_리어_M_I_RB_이상 AT %MW20030.2 : BOOL;
    R101_3축_리어_M_I_RB_자동 AT %MW20030.1 : BOOL;
    R101_3축_리어_M_I_RB_최종작업완료 AT %MW20031.0 : BOOL;
    R101_3축_리어_M_I_RB_프로그램_이상 AT %MW20030.6 : BOOL;
    R101_3축_리어_M_O_RB_1_CYCLE_SET AT %MW21030.3 : BOOL;
    R101_3축_리어_M_O_RB_1_CYCLE_리셋 AT %MW21030.4 : BOOL;
    R101_3축_리어_M_O_RB_1차_작업완료_리셋 AT %MW21032.0 : BOOL;
    R101_3축_리어_M_O_RB_2차_작업완료_리셋 AT %MW21032.1 : BOOL;
    R101_3축_리어_M_O_RB_2차_진입OK AT %MW21031.8 : BOOL;
    R101_3축_리어_M_O_RB_3차_작업완료_리셋 AT %MW21032.2 : BOOL;
    R101_3축_리어_M_O_RB_3차_진입OK AT %MW21031.9 : BOOL;
    R101_3축_리어_M_O_RB_4차_작업완료_리셋 AT %MW21032.3 : BOOL;
    R101_3축_리어_M_O_RB_4차_진입OK AT %MW21031.10 : BOOL;
    R101_3축_리어_M_O_RB_5차_작업완료_리셋 AT %MW21032.4 : BOOL;
    R101_3축_리어_M_O_RB_5차_진입OK AT %MW21031.11 : BOOL;
    R101_3축_리어_M_O_RB_6차_작업완료_리셋 AT %MW21032.5 : BOOL;
    R101_3축_리어_M_O_RB_6차_진입OK AT %MW21031.12 : BOOL;
    R101_3축_리어_M_O_RB_7차_작업완료_리셋 AT %MW21032.6 : BOOL;
    R101_3축_리어_M_O_RB_7차_진입OK AT %MW21031.13 : BOOL;
    R101_3축_리어_M_O_RB_ATD_OK AT %MW21030.6 : BOOL;
    R101_3축_리어_M_O_RB_PLT_10_진입OK AT %MW21033.10 : BOOL;
    R101_3축_리어_M_O_RB_PLT_11_진입OK AT %MW21033.11 : BOOL;
    R101_3축_리어_M_O_RB_PLT_12_진입OK AT %MW21033.12 : BOOL;
    R101_3축_리어_M_O_RB_PLT_1_진입OK AT %MW21033.1 : BOOL;
    R101_3축_리어_M_O_RB_PLT_2_진입OK AT %MW21033.2 : BOOL;
    R101_3축_리어_M_O_RB_PLT_3_진입OK AT %MW21033.3 : BOOL;
    R101_3축_리어_M_O_RB_PLT_4_진입OK AT %MW21033.4 : BOOL;
    R101_3축_리어_M_O_RB_PLT_5_진입OK AT %MW21033.5 : BOOL;
    R101_3축_리어_M_O_RB_PLT_6_진입OK AT %MW21033.6 : BOOL;
    R101_3축_리어_M_O_RB_PLT_7_진입OK AT %MW21033.7 : BOOL;
    R101_3축_리어_M_O_RB_PLT_8_진입OK AT %MW21033.8 : BOOL;
    R101_3축_리어_M_O_RB_PLT_9_진입OK AT %MW21033.9 : BOOL;
    R101_3축_리어_M_O_RB_PLT_카운터리셋_보조 AT %MW21030.10 : BOOL;
    R101_3축_리어_M_O_RB_RESTART_OK AT %MW21030.2 : BOOL;
    R101_3축_리어_M_O_RB_START_OK AT %MW21030.0 : BOOL;
    R101_3축_리어_M_O_RB_TEST_MODE_5000회 AT %MW21030.12 : BOOL;
    R101_3축_리어_M_O_RB_TIP_교체_시작 AT %MW21030.7 : BOOL;
    R101_3축_리어_M_O_RB_TIP_교체_완료 AT %MW21030.8 : BOOL;
    R101_3축_리어_M_O_RB_VIP_MODE AT %MW21030.11 : BOOL;
    R101_3축_리어_M_O_RB_냉각수_차단_요청 AT %MW21030.9 : BOOL;
    R101_3축_리어_M_O_RB_진입OK_AX차종 AT %MW21031.0 : BOOL;
    R101_3축_리어_M_O_RB_진입OK_B차종 AT %MW21031.1 : BOOL;
    R101_3축_리어_M_O_RB_진입OK_C차종 AT %MW21031.2 : BOOL;
    R101_3축_리어_M_O_RB_진입OK_D차종 AT %MW21031.3 : BOOL;
    R101_3축_리어_M_O_RB_진입OK_E차종 AT %MW21031.4 : BOOL;
    R101_3축_리어_M_O_RB_진입OK_F차종 AT %MW21031.5 : BOOL;
    R101_3축_리어_M_O_RB_진입OK_G차종 AT %MW21031.6 : BOOL;
    R101_3축_리어_M_O_RB_진입OK_H차종 AT %MW21031.7 : BOOL;
    R101_3축_리어_M_O_RB_최종_작업완료_리셋 AT %MW21030.5 : BOOL;
    R101_3축_리어_M_O_RB_프로그램_OK AT %MW21030.1 : BOOL;
    R101_3축_리어_M_RB_PROG_NO AT %MW20034 : WORD;
    R101_3축_리어_O_RB_0_5S_통신_CHK AT %MW94033.14 : BOOL;
    R101_3축_리어_O_RB_2차_진입OK AT %MW94031.8 : BOOL;
    R101_3축_리어_O_RB_3차_진입OK AT %MW94031.9 : BOOL;
    R101_3축_리어_O_RB_4차_진입OK AT %MW94031.10 : BOOL;
    R101_3축_리어_O_RB_5차_진입OK AT %MW94031.11 : BOOL;
    R101_3축_리어_O_RB_6차_진입OK AT %MW94031.12 : BOOL;
    R101_3축_리어_O_RB_7차_진입OK AT %MW94031.13 : BOOL;
    R101_3축_리어_O_RB_AX_1차_진입OK AT %MW94031.0 : BOOL;
    R101_3축_리어_O_RB_B_1차_진입OK AT %MW94031.1 : BOOL;
    R101_3축_리어_O_RB_C_1차_진입OK AT %MW94031.2 : BOOL;
    R101_3축_리어_O_RB_D_1차_진입OK AT %MW94031.3 : BOOL;
    R101_3축_리어_O_RB_EACH_작업완료_리셋 AT %MW94030.14 : BOOL;
    R101_3축_리어_O_RB_EXT_READY AT %MW94030.11 : BOOL;
    R101_3축_리어_O_RB_E_1차_진입OK AT %MW94031.4 : BOOL;
    R101_3축_리어_O_RB_F_1차_진입OK AT %MW94031.5 : BOOL;
    R101_3축_리어_O_RB_GATE_OPEN_NC AT %MW94033.11 : BOOL;
    R101_3축_리어_O_RB_G_1차_진입OK AT %MW94031.6 : BOOL;
    R101_3축_리어_O_RB_H_1차_진입OK AT %MW94031.7 : BOOL;
    R101_3축_리어_O_RB_MUTUAL_INT1 AT %MW94033.0 : BOOL;
    R101_3축_리어_O_RB_MUTUAL_INT2 AT %MW94033.1 : BOOL;
    R101_3축_리어_O_RB_MUTUAL_INT3 AT %MW94033.2 : BOOL;
    R101_3축_리어_O_RB_MUTUAL_INT4 AT %MW94033.3 : BOOL;
    R101_3축_리어_O_RB_MUTUAL_INT5 AT %MW94033.4 : BOOL;
    R101_3축_리어_O_RB_MUTUAL_INT6 AT %MW94033.5 : BOOL;
    R101_3축_리어_O_RB_MUTUAL_INT7 AT %MW94033.6 : BOOL;
    R101_3축_리어_O_RB_MUTUAL_INT8 AT %MW94033.7 : BOOL;
    R101_3축_리어_O_RB_OUTPUT AT %MW94030 : ARRAY[0..3] OF WORD;
    R101_3축_리어_O_RB_PAUSE_NC AT %MW94030.13 : BOOL;
    R101_3축_리어_O_RB_PLT10_진입OK AT %MW94032.9 : BOOL;
    R101_3축_리어_O_RB_PLT11_진입OK AT %MW94032.10 : BOOL;
    R101_3축_리어_O_RB_PLT12_진입OK AT %MW94032.11 : BOOL;
    R101_3축_리어_O_RB_PLT1_진입OK AT %MW94032.0 : BOOL;
    R101_3축_리어_O_RB_PLT2_진입OK AT %MW94032.1 : BOOL;
    R101_3축_리어_O_RB_PLT3_진입OK AT %MW94032.2 : BOOL;
    R101_3축_리어_O_RB_PLT4_진입OK AT %MW94032.3 : BOOL;
    R101_3축_리어_O_RB_PLT5_진입OK AT %MW94032.4 : BOOL;
    R101_3축_리어_O_RB_PLT6_진입OK AT %MW94032.5 : BOOL;
    R101_3축_리어_O_RB_PLT7_진입OK AT %MW94032.6 : BOOL;
    R101_3축_리어_O_RB_PLT8_진입OK AT %MW94032.7 : BOOL;
    R101_3축_리어_O_RB_PLT9_진입OK AT %MW94032.8 : BOOL;
    R101_3축_리어_O_RB_PLT_COUNT_리셋_COND AT %MW94033.10 : BOOL;
    R101_3축_리어_O_RB_PROG_선택1 AT %MW94030.0 : BOOL;
    R101_3축_리어_O_RB_PROG_선택128 AT %MW94030.7 : BOOL;
    R101_3축_리어_O_RB_PROG_선택16 AT %MW94030.4 : BOOL;
    R101_3축_리어_O_RB_PROG_선택2 AT %MW94030.1 : BOOL;
    R101_3축_리어_O_RB_PROG_선택32 AT %MW94030.5 : BOOL;
    R101_3축_리어_O_RB_PROG_선택4 AT %MW94030.2 : BOOL;
    R101_3축_리어_O_RB_PROG_선택64 AT %MW94030.6 : BOOL;
    R101_3축_리어_O_RB_PROG_선택8 AT %MW94030.3 : BOOL;
    R101_3축_리어_O_RB_SP_1_14 AT %MW94031.14 : BOOL;
    R101_3축_리어_O_RB_SP_1_15 AT %MW94031.15 : BOOL;
    R101_3축_리어_O_RB_SP_2_12 AT %MW94032.12 : BOOL;
    R101_3축_리어_O_RB_SP_2_13 AT %MW94032.13 : BOOL;
    R101_3축_리어_O_RB_SP_2_14 AT %MW94032.14 : BOOL;
    R101_3축_리어_O_RB_SP_5000TH_ON AT %MW94032.15 : BOOL;
    R101_3축_리어_O_RB_TIP_CHANGE_END AT %MW94033.9 : BOOL;
    R101_3축_리어_O_RB_TIP_CHANGE_START AT %MW94033.8 : BOOL;
    R101_3축_리어_O_RB_TIP_DRESS_SATRT AT %MW94030.12 : BOOL;
    R101_3축_리어_O_RB_VIP_MODE AT %MW94033.15 : BOOL;
    R101_3축_리어_O_RB_기동 AT %MW94030.9 : BOOL;
    R101_3축_리어_O_RB_냉각수차단 AT %MW94030.15 : BOOL;
    R101_3축_리어_O_RB_부저정지 AT %MW94033.13 : BOOL;
    R101_3축_리어_O_RB_비상정지_NC AT %MW94033.12 : BOOL;
    R101_3축_리어_O_RB_이상_리셋 AT %MW94030.10 : BOOL;
    R101_3축_리어_O_RB_작업완료_리셋 AT %MW94030.8 : BOOL;
    R101_3축_센터_I_RB_0_5_COMM_CHK AT %MW84023.14 : BOOL;
    R101_3축_센터_I_RB_10차_간섭무 AT %MW84021.9 : BOOL;
    R101_3축_센터_I_RB_11차_간섭무 AT %MW84021.10 : BOOL;
    R101_3축_센터_I_RB_12차_간섭무 AT %MW84021.11 : BOOL;
    R101_3축_센터_I_RB_1차_간섭무 AT %MW84021.0 : BOOL;
    R101_3축_센터_I_RB_1차_작업완료 AT %MW84020.9 : BOOL;
    R101_3축_센터_I_RB_2차_간섭무 AT %MW84021.1 : BOOL;
    R101_3축_센터_I_RB_2차_작업완료 AT %MW84020.10 : BOOL;
    R101_3축_센터_I_RB_3차_간섭무 AT %MW84021.2 : BOOL;
    R101_3축_센터_I_RB_3차_작업완료 AT %MW84020.11 : BOOL;
    R101_3축_센터_I_RB_4차_간섭무 AT %MW84021.3 : BOOL;
    R101_3축_센터_I_RB_4차_작업완료 AT %MW84020.12 : BOOL;
    R101_3축_센터_I_RB_5차_간섭무 AT %MW84021.4 : BOOL;
    R101_3축_센터_I_RB_5차_작업완료 AT %MW84020.13 : BOOL;
    R101_3축_센터_I_RB_6차_간섭무 AT %MW84021.5 : BOOL;
    R101_3축_센터_I_RB_6차_작업완료 AT %MW84020.14 : BOOL;
    R101_3축_센터_I_RB_7차_간섭무 AT %MW84021.6 : BOOL;
    R101_3축_센터_I_RB_7차_작업완료 AT %MW84020.15 : BOOL;
    R101_3축_센터_I_RB_8차_간섭무 AT %MW84021.7 : BOOL;
    R101_3축_센터_I_RB_9차_간섭무 AT %MW84021.8 : BOOL;
    R101_3축_센터_I_RB_AB_NORMAL_선택 AT %MW84020.6 : BOOL;
    R101_3축_센터_I_RB_GUN1_FIXED_TIP AT %MW84027 : WORD;
    R101_3축_센터_I_RB_GUN1_MOVING_TIP AT %MW84026 : WORD;
    R101_3축_센터_I_RB_GUN2_FIXED_TIP AT %MW84029 : WORD;
    R101_3축_센터_I_RB_GUN2_MOVING_TIP AT %MW84028 : WORD;
    R101_3축_센터_I_RB_INPUT AT %MW84020 : ARRAY[0..3] OF WORD;
    R101_3축_센터_I_RB_LS_이상 AT %MW84022.11 : BOOL;
    R101_3축_센터_I_RB_MOTOR_MC_ON AT %MW84023.15 : BOOL;
    R101_3축_센터_I_RB_MUTUAL_INT1 AT %MW84023.0 : BOOL;
    R101_3축_센터_I_RB_MUTUAL_INT2 AT %MW84023.1 : BOOL;
    R101_3축_센터_I_RB_MUTUAL_INT3 AT %MW84023.2 : BOOL;
    R101_3축_센터_I_RB_MUTUAL_INT4 AT %MW84023.3 : BOOL;
    R101_3축_센터_I_RB_MUTUAL_INT5 AT %MW84023.4 : BOOL;
    R101_3축_센터_I_RB_MUTUAL_INT6 AT %MW84023.5 : BOOL;
    R101_3축_센터_I_RB_MUTUAL_INT7 AT %MW84023.6 : BOOL;
    R101_3축_센터_I_RB_MUTUAL_INT8 AT %MW84023.7 : BOOL;
    R101_3축_센터_I_RB_PLT_UNLOAD_완료 AT %MW84023.11 : BOOL;
    R101_3축_센터_I_RB_PLT_최종UNLOAD_완료 AT %MW84023.12 : BOOL;
    R101_3축_센터_I_RB_PROG_ECHO_1 AT %MW84022.0 : BOOL;
    R101_3축_센터_I_RB_PROG_ECHO_128 AT %MW84022.7 : BOOL;
    R101_3축_센터_I_RB_PROG_ECHO_16 AT %MW84022.4 : BOOL;
    R101_3축_센터_I_RB_PROG_ECHO_2 AT %MW84022.1 : BOOL;
    R101_3축_센터_I_RB_PROG_ECHO_32 AT %MW84022.5 : BOOL;
    R101_3축_센터_I_RB_PROG_ECHO_4 AT %MW84022.2 : BOOL;
    R101_3축_센터_I_RB_PROG_ECHO_64 AT %MW84022.6 : BOOL;
    R101_3축_센터_I_RB_PROG_ECHO_8 AT %MW84022.3 : BOOL;
    R101_3축_센터_I_RB_SP3_8 AT %MW84023.8 : BOOL;
    R101_3축_센터_I_RB_SP3_9 AT %MW84023.9 : BOOL;
    R101_3축_센터_I_RB_SPARE_WORD_4 AT %MW84024 : WORD;
    R101_3축_센터_I_RB_SP_1_12 AT %MW84021.12 : BOOL;
    R101_3축_센터_I_RB_SP_1_13 AT %MW84021.13 : BOOL;
    R101_3축_센터_I_RB_SP_1_14 AT %MW84021.14 : BOOL;
    R101_3축_센터_I_RB_SP_1_15 AT %MW84021.15 : BOOL;
    R101_3축_센터_I_RB_TC_이상 AT %MW84022.8 : BOOL;
    R101_3축_센터_I_RB_TIP_CHANGE AT %MW84023.13 : BOOL;
    R101_3축_센터_I_RB_TIP_DRESSING AT %MW84020.7 : BOOL;
    R101_3축_센터_I_RB__PLT_카운터리셋완료 AT %MW84023.10 : BOOL;
    R101_3축_센터_I_RB_공기압_이상 AT %MW84022.9 : BOOL;
    R101_3축_센터_I_RB_냉각수_이상 AT %MW84022.10 : BOOL;
    R101_3축_센터_I_RB_비상정지_NC AT %MW84020.8 : BOOL;
    R101_3축_센터_I_RB_비전이상 AT %MW84022.14 : BOOL;
    R101_3축_센터_I_RB_실러이상 AT %MW84022.13 : BOOL;
    R101_3축_센터_I_RB_용접카운터이상 AT %MW84022.15 : BOOL;
    R101_3축_센터_I_RB_용접타점수 AT %MW84025 : WORD;
    R101_3축_센터_I_RB_운전준비 AT %MW84020.3 : BOOL;
    R101_3축_센터_I_RB_원위치 AT %MW84020.0 : BOOL;
    R101_3축_센터_I_RB_이상리셋 AT %MW84020.2 : BOOL;
    R101_3축_센터_I_RB_자동 AT %MW84020.4 : BOOL;
    R101_3축_센터_I_RB_자동기동 AT %MW84020.5 : BOOL;
    R101_3축_센터_I_RB_최종_작업완료 AT %MW84020.1 : BOOL;
    R101_3축_센터_I_RB_통신이상 AT %MW84022.12 : BOOL;
    R101_3축_센터_M_I_RB_1차_작업완료 AT %MW20021.2 : BOOL;
    R101_3축_센터_M_I_RB_2차_작업완료 AT %MW20021.3 : BOOL;
    R101_3축_센터_M_I_RB_3차_작업완료 AT %MW20021.4 : BOOL;
    R101_3축_센터_M_I_RB_4차_작업완료 AT %MW20021.5 : BOOL;
    R101_3축_센터_M_I_RB_5차_작업완료 AT %MW20021.6 : BOOL;
    R101_3축_센터_M_I_RB_6차_작업완료 AT %MW20021.7 : BOOL;
    R101_3축_센터_M_I_RB_7차_작업완료 AT %MW20021.8 : BOOL;
    R101_3축_센터_M_I_RB_PAUSE_보조 AT %MW20020.5 : BOOL;
    R101_3축_센터_M_I_RB_PLC_RUN_CHK_이상 AT %MW20020.7 : BOOL;
    R101_3축_센터_M_I_RB_간섭무_1 AT %MW20022.0 : BOOL;
    R101_3축_센터_M_I_RB_간섭무_10 AT %MW20022.9 : BOOL;
    R101_3축_센터_M_I_RB_간섭무_11 AT %MW20022.10 : BOOL;
    R101_3축_센터_M_I_RB_간섭무_12 AT %MW20022.11 : BOOL;
    R101_3축_센터_M_I_RB_간섭무_2 AT %MW20022.1 : BOOL;
    R101_3축_센터_M_I_RB_간섭무_3 AT %MW20022.2 : BOOL;
    R101_3축_센터_M_I_RB_간섭무_4 AT %MW20022.3 : BOOL;
    R101_3축_센터_M_I_RB_간섭무_5 AT %MW20022.4 : BOOL;
    R101_3축_센터_M_I_RB_간섭무_6 AT %MW20022.5 : BOOL;
    R101_3축_센터_M_I_RB_간섭무_7 AT %MW20022.6 : BOOL;
    R101_3축_센터_M_I_RB_간섭무_8 AT %MW20022.7 : BOOL;
    R101_3축_센터_M_I_RB_간섭무_9 AT %MW20022.8 : BOOL;
    R101_3축_센터_M_I_RB_비상정지 AT %MW20020.4 : BOOL;
    R101_3축_센터_M_I_RB_운전준비 AT %MW20020.0 : BOOL;
    R101_3축_센터_M_I_RB_원위치 AT %MW20020.3 : BOOL;
    R101_3축_센터_M_I_RB_이상 AT %MW20020.2 : BOOL;
    R101_3축_센터_M_I_RB_자동 AT %MW20020.1 : BOOL;
    R101_3축_센터_M_I_RB_최종작업완료 AT %MW20021.0 : BOOL;
    R101_3축_센터_M_I_RB_프로그램_이상 AT %MW20020.6 : BOOL;
    R101_3축_센터_M_O_RB_1_CYCLE_SET AT %MW21020.3 : BOOL;
    R101_3축_센터_M_O_RB_1_CYCLE_리셋 AT %MW21020.4 : BOOL;
    R101_3축_센터_M_O_RB_1차_작업완료_리셋 AT %MW21022.0 : BOOL;
    R101_3축_센터_M_O_RB_2차_작업완료_리셋 AT %MW21022.1 : BOOL;
    R101_3축_센터_M_O_RB_2차_진입OK AT %MW21021.8 : BOOL;
    R101_3축_센터_M_O_RB_3차_작업완료_리셋 AT %MW21022.2 : BOOL;
    R101_3축_센터_M_O_RB_3차_진입OK AT %MW21021.9 : BOOL;
    R101_3축_센터_M_O_RB_4차_작업완료_리셋 AT %MW21022.3 : BOOL;
    R101_3축_센터_M_O_RB_4차_진입OK AT %MW21021.10 : BOOL;
    R101_3축_센터_M_O_RB_5차_작업완료_리셋 AT %MW21022.4 : BOOL;
    R101_3축_센터_M_O_RB_5차_진입OK AT %MW21021.11 : BOOL;
    R101_3축_센터_M_O_RB_6차_작업완료_리셋 AT %MW21022.5 : BOOL;
    R101_3축_센터_M_O_RB_6차_진입OK AT %MW21021.12 : BOOL;
    R101_3축_센터_M_O_RB_7차_작업완료_리셋 AT %MW21022.6 : BOOL;
    R101_3축_센터_M_O_RB_7차_진입OK AT %MW21021.13 : BOOL;
    R101_3축_센터_M_O_RB_ATD_OK AT %MW21020.6 : BOOL;
    R101_3축_센터_M_O_RB_PLT_10_진입OK AT %MW21023.10 : BOOL;
    R101_3축_센터_M_O_RB_PLT_11_진입OK AT %MW21023.11 : BOOL;
    R101_3축_센터_M_O_RB_PLT_12_진입OK AT %MW21023.12 : BOOL;
    R101_3축_센터_M_O_RB_PLT_1_진입OK AT %MW21023.1 : BOOL;
    R101_3축_센터_M_O_RB_PLT_2_진입OK AT %MW21023.2 : BOOL;
    R101_3축_센터_M_O_RB_PLT_3_진입OK AT %MW21023.3 : BOOL;
    R101_3축_센터_M_O_RB_PLT_4_진입OK AT %MW21023.4 : BOOL;
    R101_3축_센터_M_O_RB_PLT_5_진입OK AT %MW21023.5 : BOOL;
    R101_3축_센터_M_O_RB_PLT_6_진입OK AT %MW21023.6 : BOOL;
    R101_3축_센터_M_O_RB_PLT_7_진입OK AT %MW21023.7 : BOOL;
    R101_3축_센터_M_O_RB_PLT_8_진입OK AT %MW21023.8 : BOOL;
    R101_3축_센터_M_O_RB_PLT_9_진입OK AT %MW21023.9 : BOOL;
    R101_3축_센터_M_O_RB_PLT_카운터리셋_보조 AT %MW21020.10 : BOOL;
    R101_3축_센터_M_O_RB_RESTART_OK AT %MW21020.2 : BOOL;
    R101_3축_센터_M_O_RB_START_OK AT %MW21020.0 : BOOL;
    R101_3축_센터_M_O_RB_TEST_MODE_5000회 AT %MW21020.12 : BOOL;
    R101_3축_센터_M_O_RB_TIP_교체_시작 AT %MW21020.7 : BOOL;
    R101_3축_센터_M_O_RB_TIP_교체_완료 AT %MW21020.8 : BOOL;
    R101_3축_센터_M_O_RB_VIP_MODE AT %MW21020.11 : BOOL;
    R101_3축_센터_M_O_RB_냉각수_차단_요청 AT %MW21020.9 : BOOL;
    R101_3축_센터_M_O_RB_진입OK_AX차종 AT %MW21021.0 : BOOL;
    R101_3축_센터_M_O_RB_진입OK_B차종 AT %MW21021.1 : BOOL;
    R101_3축_센터_M_O_RB_진입OK_C차종 AT %MW21021.2 : BOOL;
    R101_3축_센터_M_O_RB_진입OK_D차종 AT %MW21021.3 : BOOL;
    R101_3축_센터_M_O_RB_진입OK_E차종 AT %MW21021.4 : BOOL;
    R101_3축_센터_M_O_RB_진입OK_F차종 AT %MW21021.5 : BOOL;
    R101_3축_센터_M_O_RB_진입OK_G차종 AT %MW21021.6 : BOOL;
    R101_3축_센터_M_O_RB_진입OK_H차종 AT %MW21021.7 : BOOL;
    R101_3축_센터_M_O_RB_최종_작업완료_리셋 AT %MW21020.5 : BOOL;
    R101_3축_센터_M_O_RB_프로그램_OK AT %MW21020.1 : BOOL;
    R101_3축_센터_M_RB_PROG_NO AT %MW20024 : WORD;
    R101_3축_센터_O_RB_0_5S_통신_CHK AT %MW94023.14 : BOOL;
    R101_3축_센터_O_RB_2차_진입OK AT %MW94021.8 : BOOL;
    R101_3축_센터_O_RB_3차_진입OK AT %MW94021.9 : BOOL;
    R101_3축_센터_O_RB_4차_진입OK AT %MW94021.10 : BOOL;
    R101_3축_센터_O_RB_5차_진입OK AT %MW94021.11 : BOOL;
    R101_3축_센터_O_RB_6차_진입OK AT %MW94021.12 : BOOL;
    R101_3축_센터_O_RB_7차_진입OK AT %MW94021.13 : BOOL;
    R101_3축_센터_O_RB_AX_1차_진입OK AT %MW94021.0 : BOOL;
    R101_3축_센터_O_RB_B_1차_진입OK AT %MW94021.1 : BOOL;
    R101_3축_센터_O_RB_C_1차_진입OK AT %MW94021.2 : BOOL;
    R101_3축_센터_O_RB_D_1차_진입OK AT %MW94021.3 : BOOL;
    R101_3축_센터_O_RB_EACH_작업완료_리셋 AT %MW94020.14 : BOOL;
    R101_3축_센터_O_RB_EXT_READY AT %MW94020.11 : BOOL;
    R101_3축_센터_O_RB_E_1차_진입OK AT %MW94021.4 : BOOL;
    R101_3축_센터_O_RB_F_1차_진입OK AT %MW94021.5 : BOOL;
    R101_3축_센터_O_RB_GATE_OPEN_NC AT %MW94023.11 : BOOL;
    R101_3축_센터_O_RB_G_1차_진입OK AT %MW94021.6 : BOOL;
    R101_3축_센터_O_RB_H_1차_진입OK AT %MW94021.7 : BOOL;
    R101_3축_센터_O_RB_MUTUAL_INT1 AT %MW94023.0 : BOOL;
    R101_3축_센터_O_RB_MUTUAL_INT2 AT %MW94023.1 : BOOL;
    R101_3축_센터_O_RB_MUTUAL_INT3 AT %MW94023.2 : BOOL;
    R101_3축_센터_O_RB_MUTUAL_INT4 AT %MW94023.3 : BOOL;
    R101_3축_센터_O_RB_MUTUAL_INT5 AT %MW94023.4 : BOOL;
    R101_3축_센터_O_RB_MUTUAL_INT6 AT %MW94023.5 : BOOL;
    R101_3축_센터_O_RB_MUTUAL_INT7 AT %MW94023.6 : BOOL;
    R101_3축_센터_O_RB_MUTUAL_INT8 AT %MW94023.7 : BOOL;
    R101_3축_센터_O_RB_OUTPUT AT %MW94020 : ARRAY[0..3] OF WORD;
    R101_3축_센터_O_RB_PAUSE_NC AT %MW94020.13 : BOOL;
    R101_3축_센터_O_RB_PLT10_진입OK AT %MW94022.9 : BOOL;
    R101_3축_센터_O_RB_PLT11_진입OK AT %MW94022.10 : BOOL;
    R101_3축_센터_O_RB_PLT12_진입OK AT %MW94022.11 : BOOL;
    R101_3축_센터_O_RB_PLT1_진입OK AT %MW94022.0 : BOOL;
    R101_3축_센터_O_RB_PLT2_진입OK AT %MW94022.1 : BOOL;
    R101_3축_센터_O_RB_PLT3_진입OK AT %MW94022.2 : BOOL;
    R101_3축_센터_O_RB_PLT4_진입OK AT %MW94022.3 : BOOL;
    R101_3축_센터_O_RB_PLT5_진입OK AT %MW94022.4 : BOOL;
    R101_3축_센터_O_RB_PLT6_진입OK AT %MW94022.5 : BOOL;
    R101_3축_센터_O_RB_PLT7_진입OK AT %MW94022.6 : BOOL;
    R101_3축_센터_O_RB_PLT8_진입OK AT %MW94022.7 : BOOL;
    R101_3축_센터_O_RB_PLT9_진입OK AT %MW94022.8 : BOOL;
    R101_3축_센터_O_RB_PLT_COUNT_리셋_COND AT %MW94023.10 : BOOL;
    R101_3축_센터_O_RB_PROG_선택1 AT %MW94020.0 : BOOL;
    R101_3축_센터_O_RB_PROG_선택128 AT %MW94020.7 : BOOL;
    R101_3축_센터_O_RB_PROG_선택16 AT %MW94020.4 : BOOL;
    R101_3축_센터_O_RB_PROG_선택2 AT %MW94020.1 : BOOL;
    R101_3축_센터_O_RB_PROG_선택32 AT %MW94020.5 : BOOL;
    R101_3축_센터_O_RB_PROG_선택4 AT %MW94020.2 : BOOL;
    R101_3축_센터_O_RB_PROG_선택64 AT %MW94020.6 : BOOL;
    R101_3축_센터_O_RB_PROG_선택8 AT %MW94020.3 : BOOL;
    R101_3축_센터_O_RB_SP_1_14 AT %MW94021.14 : BOOL;
    R101_3축_센터_O_RB_SP_1_15 AT %MW94021.15 : BOOL;
    R101_3축_센터_O_RB_SP_2_12 AT %MW94022.12 : BOOL;
    R101_3축_센터_O_RB_SP_2_13 AT %MW94022.13 : BOOL;
    R101_3축_센터_O_RB_SP_2_14 AT %MW94022.14 : BOOL;
    R101_3축_센터_O_RB_SP_5000TH_ON AT %MW94022.15 : BOOL;
    R101_3축_센터_O_RB_TIP_CHANGE_END AT %MW94023.9 : BOOL;
    R101_3축_센터_O_RB_TIP_CHANGE_START AT %MW94023.8 : BOOL;
    R101_3축_센터_O_RB_TIP_DRESS_SATRT AT %MW94020.12 : BOOL;
    R101_3축_센터_O_RB_VIP_MODE AT %MW94023.15 : BOOL;
    R101_3축_센터_O_RB_기동 AT %MW94020.9 : BOOL;
    R101_3축_센터_O_RB_냉각수차단 AT %MW94020.15 : BOOL;
    R101_3축_센터_O_RB_부저정지 AT %MW94023.13 : BOOL;
    R101_3축_센터_O_RB_비상정지_NC AT %MW94023.12 : BOOL;
    R101_3축_센터_O_RB_이상_리셋 AT %MW94020.10 : BOOL;
    R101_3축_센터_O_RB_작업완료_리셋 AT %MW94020.8 : BOOL;
    R101_3축_프론트_I_RB_0_5_COMM_CHK AT %MW84013.14 : BOOL;
    R101_3축_프론트_I_RB_10차_간섭무 AT %MW84011.9 : BOOL;
    R101_3축_프론트_I_RB_11차_간섭무 AT %MW84011.10 : BOOL;
    R101_3축_프론트_I_RB_12차_간섭무 AT %MW84011.11 : BOOL;
    R101_3축_프론트_I_RB_1차_간섭무 AT %MW84011.0 : BOOL;
    R101_3축_프론트_I_RB_1차_작업완료 AT %MW84010.9 : BOOL;
    R101_3축_프론트_I_RB_2차_간섭무 AT %MW84011.1 : BOOL;
    R101_3축_프론트_I_RB_2차_작업완료 AT %MW84010.10 : BOOL;
    R101_3축_프론트_I_RB_3차_간섭무 AT %MW84011.2 : BOOL;
    R101_3축_프론트_I_RB_3차_작업완료 AT %MW84010.11 : BOOL;
    R101_3축_프론트_I_RB_4차_간섭무 AT %MW84011.3 : BOOL;
    R101_3축_프론트_I_RB_4차_작업완료 AT %MW84010.12 : BOOL;
    R101_3축_프론트_I_RB_5차_간섭무 AT %MW84011.4 : BOOL;
    R101_3축_프론트_I_RB_5차_작업완료 AT %MW84010.13 : BOOL;
    R101_3축_프론트_I_RB_6차_간섭무 AT %MW84011.5 : BOOL;
    R101_3축_프론트_I_RB_6차_작업완료 AT %MW84010.14 : BOOL;
    R101_3축_프론트_I_RB_7차_간섭무 AT %MW84011.6 : BOOL;
    R101_3축_프론트_I_RB_7차_작업완료 AT %MW84010.15 : BOOL;
    R101_3축_프론트_I_RB_8차_간섭무 AT %MW84011.7 : BOOL;
    R101_3축_프론트_I_RB_9차_간섭무 AT %MW84011.8 : BOOL;
    R101_3축_프론트_I_RB_AB_NORMAL_선택 AT %MW84010.6 : BOOL;
    R101_3축_프론트_I_RB_GUN1_FIXED_TIP AT %MW84017 : WORD;
    R101_3축_프론트_I_RB_GUN1_MOVING_TIP AT %MW84016 : WORD;
    R101_3축_프론트_I_RB_GUN2_FIXED_TIP AT %MW84019 : WORD;
    R101_3축_프론트_I_RB_GUN2_MOVING_TIP AT %MW84018 : WORD;
    R101_3축_프론트_I_RB_INPUT AT %MW84010 : ARRAY[0..3] OF WORD;
    R101_3축_프론트_I_RB_LS_이상 AT %MW84012.11 : BOOL;
    R101_3축_프론트_I_RB_MOTOR_MC_ON AT %MW84013.15 : BOOL;
    R101_3축_프론트_I_RB_MUTUAL_INT1 AT %MW84013.0 : BOOL;
    R101_3축_프론트_I_RB_MUTUAL_INT2 AT %MW84013.1 : BOOL;
    R101_3축_프론트_I_RB_MUTUAL_INT3 AT %MW84013.2 : BOOL;
    R101_3축_프론트_I_RB_MUTUAL_INT4 AT %MW84013.3 : BOOL;
    R101_3축_프론트_I_RB_MUTUAL_INT5 AT %MW84013.4 : BOOL;
    R101_3축_프론트_I_RB_MUTUAL_INT6 AT %MW84013.5 : BOOL;
    R101_3축_프론트_I_RB_MUTUAL_INT7 AT %MW84013.6 : BOOL;
    R101_3축_프론트_I_RB_MUTUAL_INT8 AT %MW84013.7 : BOOL;
    R101_3축_프론트_I_RB_PLT_UNLOAD_완료 AT %MW84013.11 : BOOL;
    R101_3축_프론트_I_RB_PLT_최종UNLOAD_완료 AT %MW84013.12 : BOOL;
    R101_3축_프론트_I_RB_PROG_ECHO_1 AT %MW84012.0 : BOOL;
    R101_3축_프론트_I_RB_PROG_ECHO_128 AT %MW84012.7 : BOOL;
    R101_3축_프론트_I_RB_PROG_ECHO_16 AT %MW84012.4 : BOOL;
    R101_3축_프론트_I_RB_PROG_ECHO_2 AT %MW84012.1 : BOOL;
    R101_3축_프론트_I_RB_PROG_ECHO_32 AT %MW84012.5 : BOOL;
    R101_3축_프론트_I_RB_PROG_ECHO_4 AT %MW84012.2 : BOOL;
    R101_3축_프론트_I_RB_PROG_ECHO_64 AT %MW84012.6 : BOOL;
